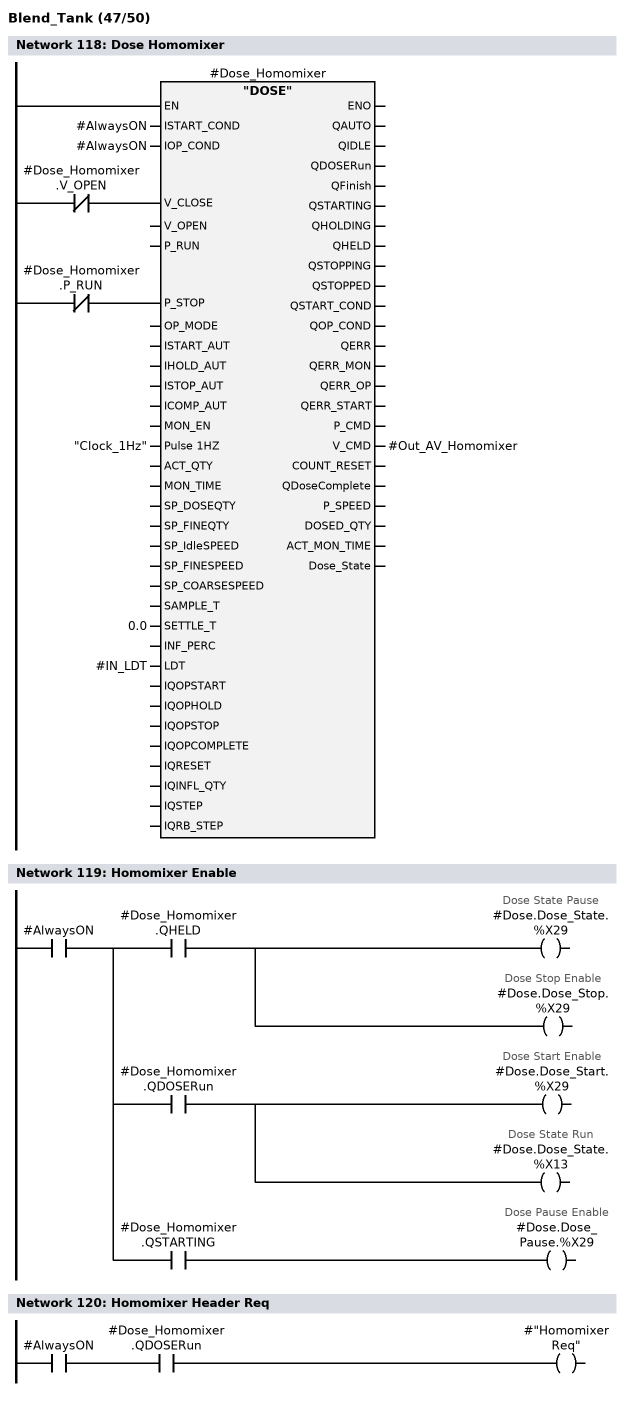
   RUNG wire#powerrail
      #Dose_Homomixer(V_CLOSE := wire#w1, P_STOP := wire#w2, ISTART_COND := #AlwaysON, IOP_COND := #AlwaysON, V_OPEN :=, P_RUN :=, OP_MODE :=, ISTART_AUT :=, IHOLD_AUT :=, ISTOP_AUT :=, ICOMP_AUT :=, MON_EN :=, "Pulse 1HZ" := "Clock_1Hz", ACT_QTY :=, MON_TIME :=, SP_DOSEQTY :=, SP_FINEQTY :=, SP_IdleSPEED :=, SP_FINESPEED :=, SP_COARSESPEED :=, SAMPLE_T :=, SETTLE_T := 0.0, INF_PERC :=, LDT := #IN_LDT, IQOPSTART :=, IQOPHOLD :=, IQOPSTOP :=, IQOPCOMPLETE :=, IQRESET :=, IQINFL_QTY :=, IQSTEP :=, IQRB_STEP :=, QAUTO =>, QIDLE =>, QDOSERun =>, QFinish =>, QSTARTING =>, QHOLDING =>, QHELD =>, QSTOPPING =>, QSTOPPED =>, QSTART_COND =>, QOP_COND =>, QERR =>, QERR_MON =>, QERR_OP =>, QERR_START =>, P_CMD =>, V_CMD => #Out_AV_Homomixer, COUNT_RESET =>, QDoseComplete =>, P_SPEED =>, DOSED_QTY =>, ACT_MON_TIME =>, Dose_State =>)
   END_RUNG
   RUNG wire#powerrail
      I_Contact( #Dose_Homomixer.V_OPEN )
   END_RUNG wire#w1
   RUNG wire#powerrail
      I_Contact( #Dose_Homomixer.P_RUN )
   END_RUNG wire#w2
   // the same network as SCL:
   #Dose_Homomixer(ISTART_COND := #AlwaysON,   // "DOSE"
                   IOP_COND := #AlwaysON,
                   V_CLOSE := NOT #Dose_Homomixer.V_OPEN,
                   P_STOP := NOT #Dose_Homomixer.P_RUN,
                   "Pulse 1HZ" := "Clock_1Hz",
                   SETTLE_T := 0.0,
                   LDT := #IN_LDT,
                   V_CMD => #Out_AV_Homomixer);
END_REGION

REGION Network 119: Homomixer Enable
   RUNG wire#powerrail
      Contact( #AlwaysON )
      wire#w1
      Contact( #Dose_Homomixer.QHELD )
      wire#w2
      Coil( #Dose.Dose_State.%X29 )   // Dose State Pause
   END_RUNG
   RUNG wire#w2
      Coil( #Dose.Dose_Stop.%X29 )   // Dose Stop Enable
   END_RUNG
   RUNG wire#w1
      Contact( #Dose_Homomixer.QDOSERun )
      wire#w3
      Coil( #Dose.Dose_Start.%X29 )   // Dose Start Enable
   END_RUNG
   RUNG wire#w3
      Coil( #Dose.Dose_State.%X13 )   // Dose State Run
   END_RUNG
   RUNG wire#w1
      Contact( #Dose_Homomixer.QSTARTING )
      Coil( #Dose.Dose_Pause.%X29 )   // Dose Pause Enable
   END_RUNG
   // the same network as SCL:
   #Dose.Dose_State.%X29 := #AlwaysON AND #Dose_Homomixer.QHELD;   // Dose State Pause
   #Dose.Dose_Stop.%X29 := #Dose.Dose_State.%X29;   // Dose Stop Enable
   #Dose.Dose_Start.%X29 := #AlwaysON AND #Dose_Homomixer.QDOSERun;   // Dose Start Enable
   #Dose.Dose_State.%X13 := #Dose.Dose_Start.%X29;   // Dose State Run
   #Dose.Dose_Pause.%X29 := #AlwaysON AND #Dose_Homomixer.QSTARTING;   // Dose Pause Enable
END_REGION

REGION Network 120: Homomixer Header Req
   RUNG wire#powerrail
      Contact( #AlwaysON )
      Contact( #Dose_Homomixer.QDOSERun )
      Coil( #"Homomixer Req" )
   END_RUNG
   // the same network as SCL:
   #"Homomixer Req" := #AlwaysON AND #Dose_Homomixer.QDOSERun;
END_REGION

REGION Network 122: Level Scaling
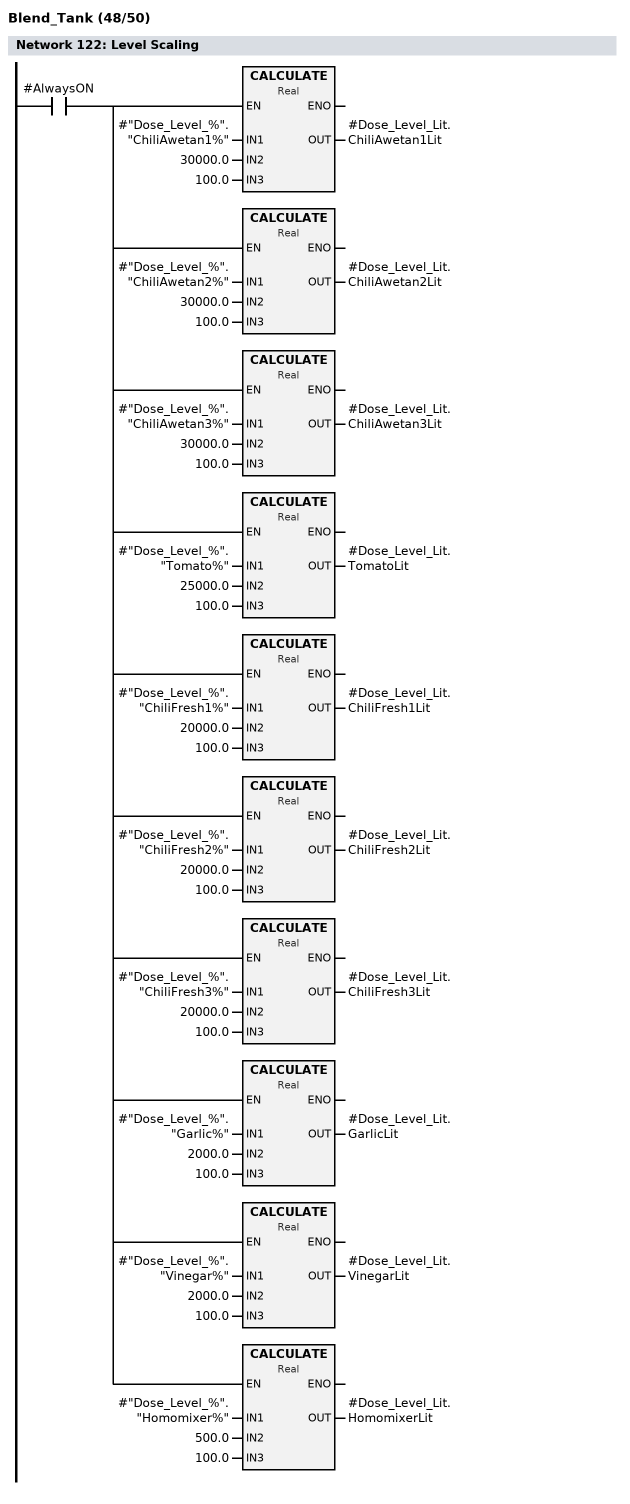
   RUNG wire#powerrail
      Contact( #AlwaysON )
      wire#w1
      { S7_Templates := "SrcType := Real"; S7_Expression := "(IN1 * IN2) / IN3" } Calculate(in1 := #"Dose_Level_%"."ChiliAwetan1%", in2 := 30000.0, in3 := 100.0, out => #Dose_Level_Lit.ChiliAwetan1Lit)
   END_RUNG
   RUNG wire#w1
      { S7_Templates := "SrcType := Real"; S7_Expression := "(IN1 * IN2) / IN3" } Calculate(in1 := #"Dose_Level_%"."ChiliAwetan2%", in2 := 30000.0, in3 := 100.0, out => #Dose_Level_Lit.ChiliAwetan2Lit)
   END_RUNG
   RUNG wire#w1
      { S7_Templates := "SrcType := Real"; S7_Expression := "(IN1 * IN2) / IN3" } Calculate(in1 := #"Dose_Level_%"."ChiliAwetan3%", in2 := 30000.0, in3 := 100.0, out => #Dose_Level_Lit.ChiliAwetan3Lit)
   END_RUNG
   RUNG wire#w1
      { S7_Templates := "SrcType := Real"; S7_Expression := "(IN1 * IN2) / IN3" } Calculate(in1 := #"Dose_Level_%"."Tomato%", in2 := 25000.0, in3 := 100.0, out => #Dose_Level_Lit.TomatoLit)
   END_RUNG
   RUNG wire#w1
      { S7_Templates := "SrcType := Real"; S7_Expression := "(IN1 * IN2) / IN3" } Calculate(in1 := #"Dose_Level_%"."ChiliFresh1%", in2 := 20000.0, in3 := 100.0, out => #Dose_Level_Lit.ChiliFresh1Lit)
   END_RUNG
   RUNG wire#w1
      { S7_Templates := "SrcType := Real"; S7_Expression := "(IN1 * IN2) / IN3" } Calculate(in1 := #"Dose_Level_%"."ChiliFresh2%", in2 := 20000.0, in3 := 100.0, out => #Dose_Level_Lit.ChiliFresh2Lit)
   END_RUNG
   RUNG wire#w1
      { S7_Templates := "SrcType := Real"; S7_Expression := "(IN1 * IN2) / IN3" } Calculate(in1 := #"Dose_Level_%"."ChiliFresh3%", in2 := 20000.0, in3 := 100.0, out => #Dose_Level_Lit.ChiliFresh3Lit)
   END_RUNG
   RUNG wire#w1
      { S7_Templates := "SrcType := Real"; S7_Expression := "(IN1 * IN2) / IN3" } Calculate(in1 := #"Dose_Level_%"."Garlic%", in2 := 2000.0, in3 := 100.0, out => #Dose_Level_Lit.GarlicLit)
   END_RUNG
   RUNG wire#w1
      { S7_Templates := "SrcType := Real"; S7_Expression := "(IN1 * IN2) / IN3" } Calculate(in1 := #"Dose_Level_%"."Vinegar%", in2 := 2000.0, in3 := 100.0, out => #Dose_Level_Lit.VinegarLit)
   END_RUNG
   RUNG wire#w1
      { S7_Templates := "SrcType := Real"; S7_Expression := "(IN1 * IN2) / IN3" } Calculate(in1 := #"Dose_Level_%"."Homomixer%", in2 := 500.0, in3 := 100.0, out => #Dose_Level_Lit.HomomixerLit)
   END_RUNG
   // the same network as SCL:
   IF #AlwaysON THEN
       #Dose_Level_Lit.ChiliAwetan1Lit := (#"Dose_Level_%"."ChiliAwetan1%" * 30000.0) / 100.0;
       #Dose_Level_Lit.ChiliAwetan2Lit := (#"Dose_Level_%"."ChiliAwetan2%" * 30000.0) / 100.0;
       #Dose_Level_Lit.ChiliAwetan3Lit := (#"Dose_Level_%"."ChiliAwetan3%" * 30000.0) / 100.0;
       #Dose_Level_Lit.TomatoLit := (#"Dose_Level_%"."Tomato%" * 25000.0) / 100.0;
       #Dose_Level_Lit.ChiliFresh1Lit := (#"Dose_Level_%"."ChiliFresh1%" * 20000.0) / 100.0;
       #Dose_Level_Lit.ChiliFresh2Lit := (#"Dose_Level_%"."ChiliFresh2%" * 20000.0) / 100.0;
       #Dose_Level_Lit.ChiliFresh3Lit := (#"Dose_Level_%"."ChiliFresh3%" * 20000.0) / 100.0;
       #Dose_Level_Lit.GarlicLit := (#"Dose_Level_%"."Garlic%" * 2000.0) / 100.0;
       #Dose_Level_Lit.VinegarLit := (#"Dose_Level_%"."Vinegar%" * 2000.0) / 100.0;
       #Dose_Level_Lit.HomomixerLit := (#"Dose_Level_%"."Homomixer%" * 500.0) / 100.0;
   END_IF;
END_REGION

REGION Network 123: Last Dose Qty
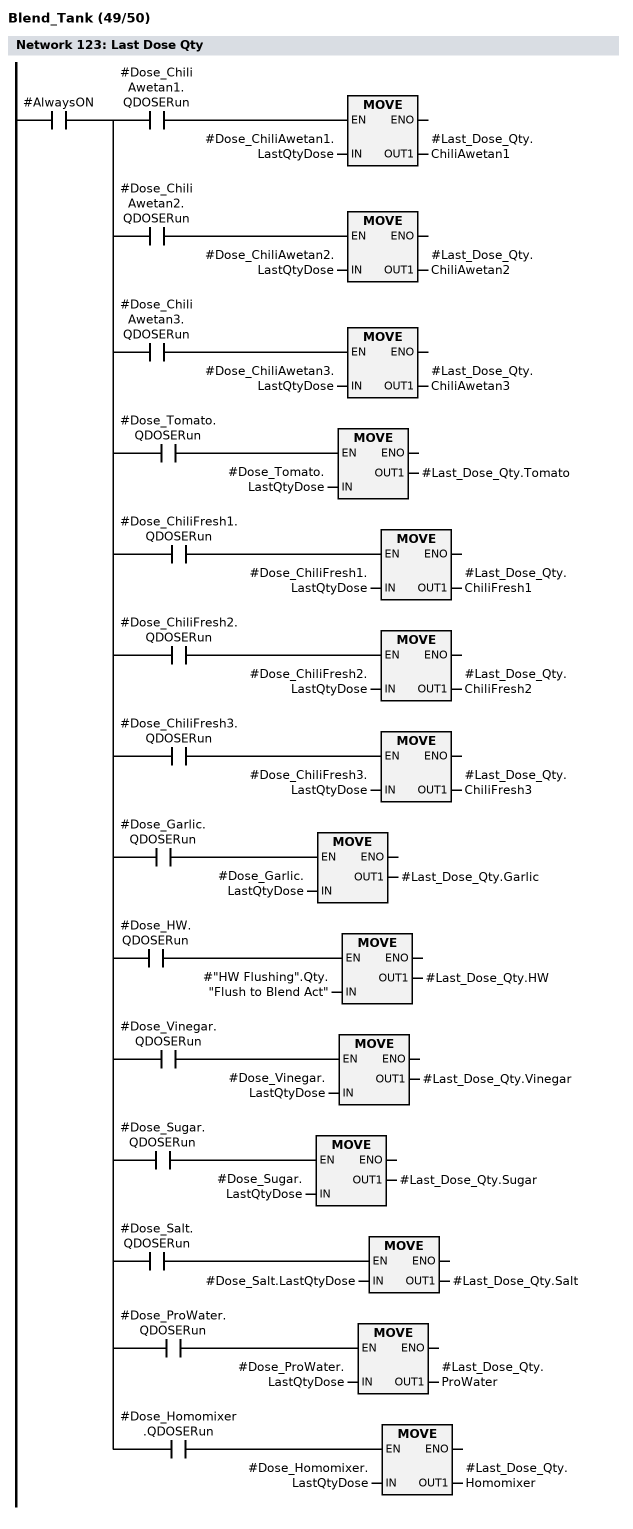
   RUNG wire#powerrail
      Contact( #AlwaysON )
      wire#w1
      Contact( #Dose_ChiliAwetan1.QDOSERun )
      Move(in := #Dose_ChiliAwetan1.LastQtyDose, out1 => #Last_Dose_Qty.ChiliAwetan1)
   END_RUNG
   RUNG wire#w1
      Contact( #Dose_ChiliAwetan2.QDOSERun )
      Move(in := #Dose_ChiliAwetan2.LastQtyDose, out1 => #Last_Dose_Qty.ChiliAwetan2)
   END_RUNG
   RUNG wire#w1
      Contact( #Dose_ChiliAwetan3.QDOSERun )
      Move(in := #Dose_ChiliAwetan3.LastQtyDose, out1 => #Last_Dose_Qty.ChiliAwetan3)
   END_RUNG
   RUNG wire#w1
      Contact( #Dose_Tomato.QDOSERun )
      Move(in := #Dose_Tomato.LastQtyDose, out1 => #Last_Dose_Qty.Tomato)
   END_RUNG
   RUNG wire#w1
      Contact( #Dose_ChiliFresh1.QDOSERun )
      Move(in := #Dose_ChiliFresh1.LastQtyDose, out1 => #Last_Dose_Qty.ChiliFresh1)
   END_RUNG
   RUNG wire#w1
      Contact( #Dose_ChiliFresh2.QDOSERun )
      Move(in := #Dose_ChiliFresh2.LastQtyDose, out1 => #Last_Dose_Qty.ChiliFresh2)
   END_RUNG
   RUNG wire#w1
      Contact( #Dose_ChiliFresh3.QDOSERun )
      Move(in := #Dose_ChiliFresh3.LastQtyDose, out1 => #Last_Dose_Qty.ChiliFresh3)
   END_RUNG
   RUNG wire#w1
      Contact( #Dose_Garlic.QDOSERun )
      Move(in := #Dose_Garlic.LastQtyDose, out1 => #Last_Dose_Qty.Garlic)
   END_RUNG
   RUNG wire#w1
      Contact( #Dose_HW.QDOSERun )
      Move(in := #"HW Flushing".Qty."Flush to Blend Act", out1 => #Last_Dose_Qty.HW)
   END_RUNG
   RUNG wire#w1
      Contact( #Dose_Vinegar.QDOSERun )
      Move(in := #Dose_Vinegar.LastQtyDose, out1 => #Last_Dose_Qty.Vinegar)
   END_RUNG
   RUNG wire#w1
      Contact( #Dose_Sugar.QDOSERun )
      Move(in := #Dose_Sugar.LastQtyDose, out1 => #Last_Dose_Qty.Sugar)
   END_RUNG
   RUNG wire#w1
      Contact( #Dose_Salt.QDOSERun )
      Move(in := #Dose_Salt.LastQtyDose, out1 => #Last_Dose_Qty.Salt)
   END_RUNG
   RUNG wire#w1
      Contact( #Dose_ProWater.QDOSERun )
      Move(in := #Dose_ProWater.LastQtyDose, out1 => #Last_Dose_Qty.ProWater)
   END_RUNG
   RUNG wire#w1
      Contact( #Dose_Homomixer.QDOSERun )
      Move(in := #Dose_Homomixer.LastQtyDose, out1 => #Last_Dose_Qty.Homomixer)
   END_RUNG
   // the same network as SCL:
   IF #AlwaysON AND #Dose_ChiliAwetan1.QDOSERun THEN
       #Last_Dose_Qty.ChiliAwetan1 := #Dose_ChiliAwetan1.LastQtyDose;
   END_IF;
   IF #AlwaysON AND #Dose_ChiliAwetan2.QDOSERun THEN
       #Last_Dose_Qty.ChiliAwetan2 := #Dose_ChiliAwetan2.LastQtyDose;
   END_IF;
   IF #AlwaysON AND #Dose_ChiliAwetan3.QDOSERun THEN
       #Last_Dose_Qty.ChiliAwetan3 := #Dose_ChiliAwetan3.LastQtyDose;
   END_IF;
   IF #AlwaysON AND #Dose_Tomato.QDOSERun THEN #Last_Dose_Qty.Tomato := #Dose_Tomato.LastQtyDose; END_IF;
   IF #AlwaysON AND #Dose_ChiliFresh1.QDOSERun THEN
       #Last_Dose_Qty.ChiliFresh1 := #Dose_ChiliFresh1.LastQtyDose;
   END_IF;
   IF #AlwaysON AND #Dose_ChiliFresh2.QDOSERun THEN
       #Last_Dose_Qty.ChiliFresh2 := #Dose_ChiliFresh2.LastQtyDose;
   END_IF;
   IF #AlwaysON AND #Dose_ChiliFresh3.QDOSERun THEN
       #Last_Dose_Qty.ChiliFresh3 := #Dose_ChiliFresh3.LastQtyDose;
   END_IF;
   IF #AlwaysON AND #Dose_Garlic.QDOSERun THEN #Last_Dose_Qty.Garlic := #Dose_Garlic.LastQtyDose; END_IF;
   IF #AlwaysON AND #Dose_HW.QDOSERun THEN
       #Last_Dose_Qty.HW := #"HW Flushing".Qty."Flush to Blend Act";
   END_IF;
   IF #AlwaysON AND #Dose_Vinegar.QDOSERun THEN #Last_Dose_Qty.Vinegar := #Dose_Vinegar.LastQtyDose; END_IF;
   IF #AlwaysON AND #Dose_Sugar.QDOSERun THEN #Last_Dose_Qty.Sugar := #Dose_Sugar.LastQtyDose; END_IF;
   IF #AlwaysON AND #Dose_Salt.QDOSERun THEN #Last_Dose_Qty.Salt := #Dose_Salt.LastQtyDose; END_IF;
   IF #AlwaysON AND #Dose_ProWater.QDOSERun THEN
       #Last_Dose_Qty.ProWater := #Dose_ProWater.LastQtyDose;
   END_IF;
   IF #AlwaysON AND #Dose_Homomixer.QDOSERun THEN
       #Last_Dose_Qty.Homomixer := #Dose_Homomixer.LastQtyDose;
   END_IF;
END_REGION

REGION Network 124: Reset Last Dose Qty After CIP Tank
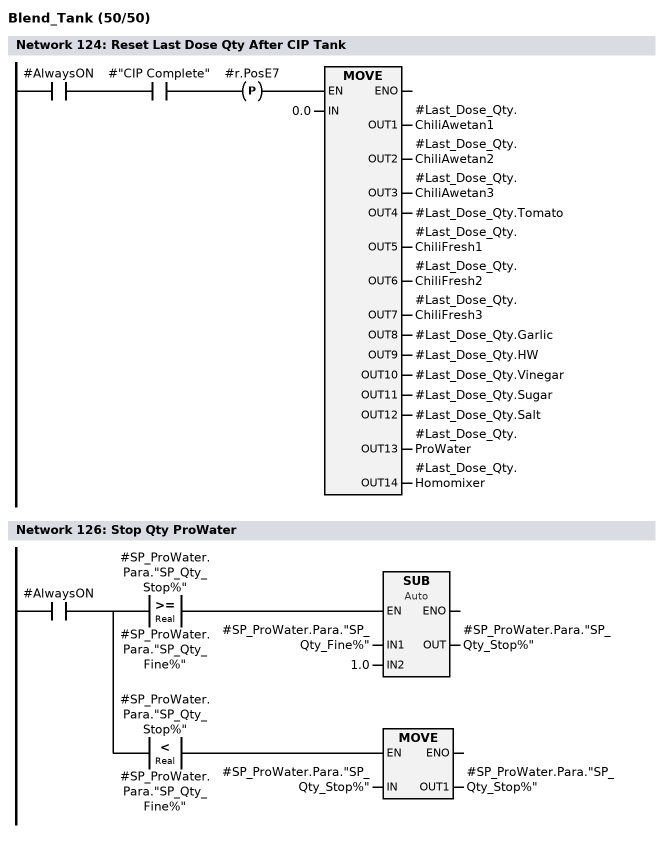
   RUNG wire#powerrail
      Contact( #AlwaysON )
      Contact( #"CIP Complete" )
      P_Trig( #r.PosE7 )
      Move(in := 0.0, out1 => #Last_Dose_Qty.ChiliAwetan1, out2 => #Last_Dose_Qty.ChiliAwetan2, out3 => #Last_Dose_Qty.ChiliAwetan3, out4 => #Last_Dose_Qty.Tomato, out5 => #Last_Dose_Qty.ChiliFresh1, out6 => #Last_Dose_Qty.ChiliFresh2, out7 => #Last_Dose_Qty.ChiliFresh3, out8 => #Last_Dose_Qty.Garlic, out9 => #Last_Dose_Qty.HW, out10 => #Last_Dose_Qty.Vinegar, out11 => #Last_Dose_Qty.Sugar, out12 => #Last_Dose_Qty.Salt, out13 => #Last_Dose_Qty.ProWater, out14 => #Last_Dose_Qty.Homomixer)
   END_RUNG
   // the same network as SCL:
   #_w1 := #AlwaysON AND #"CIP Complete";
   #_w2 := #_w1 AND NOT #r.PosE7;   // rising edge
   #r.PosE7 := #_w1;
   IF #_w2 THEN
       #Last_Dose_Qty.ChiliAwetan1 := 0.0;
       #Last_Dose_Qty.ChiliAwetan2 := 0.0;
       #Last_Dose_Qty.ChiliAwetan3 := 0.0;
       #Last_Dose_Qty.Tomato := 0.0;
       #Last_Dose_Qty.ChiliFresh1 := 0.0;
       #Last_Dose_Qty.ChiliFresh2 := 0.0;
       #Last_Dose_Qty.ChiliFresh3 := 0.0;
       #Last_Dose_Qty.Garlic := 0.0;
       #Last_Dose_Qty.HW := 0.0;
       #Last_Dose_Qty.Vinegar := 0.0;
       #Last_Dose_Qty.Sugar := 0.0;
       #Last_Dose_Qty.Salt := 0.0;
       #Last_Dose_Qty.ProWater := 0.0;
       #Last_Dose_Qty.Homomixer := 0.0;
   END_IF;
END_REGION

REGION Network 126: Stop Qty ProWater
   RUNG wire#powerrail
      Contact( #AlwaysON )
      wire#w1
      { S7_Templates := "SrcType := Real" } GE_Contact(in1 := #SP_ProWater.Para."SP_Qty_Stop%", in2 := #SP_ProWater.Para."SP_Qty_Fine%")
      Sub(in1 := #SP_ProWater.Para."SP_Qty_Fine%", in2 := 1.0, out => #SP_ProWater.Para."SP_Qty_Stop%")
   END_RUNG
   RUNG wire#w1
      { S7_Templates := "SrcType := Real" } LT_Contact(in1 := #SP_ProWater.Para."SP_Qty_Stop%", in2 := #SP_ProWater.Para."SP_Qty_Fine%")
      Move(in := #SP_ProWater.Para."SP_Qty_Stop%", out1 => #SP_ProWater.Para."SP_Qty_Stop%")
   END_RUNG
   // the same network as SCL:
   IF #AlwaysON AND (#SP_ProWater.Para."SP_Qty_Stop%" >= #SP_ProWater.Para."SP_Qty_Fine%") THEN
       #SP_ProWater.Para."SP_Qty_Stop%" := #SP_ProWater.Para."SP_Qty_Fine%" - 1.0;
   END_IF;
   IF #AlwaysON AND (#SP_ProWater.Para."SP_Qty_Stop%" < #SP_ProWater.Para."SP_Qty_Fine%") THEN
       #SP_ProWater.Para."SP_Qty_Stop%" := #SP_ProWater.Para."SP_Qty_Stop%";
   END_IF;
END_REGION
END_FUNCTION_BLOCK

FUNCTION_BLOCK "IO_Valve_Blend20"   // FB24, LAD
{ S7_Optimized_Access := 'FALSE' }
VERSION : 0.1
// stored: AutoNumber true, IsIECCheckEnabled false, SetENOAutomatically false, UDAEnableTagReadback false
   VAR_INPUT
      "lock 1" : Bool;
      "lock 2" : Bool;
      "lock 3" : Bool;
      "lock 4" : Bool;
      init : Bool;
      reset : Bool;
      testing : Bool;
   END_VAR
   VAR
      "AV-20.01" : "Valve";
      "AV-20.02" : "Valve";
      "AV-20.03" : "Valve";
      "AV-20.04" : "Valve";
      "AV-20.05" : "Valve";
      "AV-20.06" : "Valve";
      "AV-20.07" : "Valve";
      "AV-20.08" : "Valve";
      "AV-20.09" : "Valve";
      "AV-20.10" : "Valve";
      "AV-20.11" : "Valve";
      "AV-20.21" : "Valve";
      "AV-20.22" : "Valve";
      "AV-20.23" : "Valve";
      "AV-20.24" : "Valve";
      "AV-20.25" : "Valve";
      "AV-20.26" : "Valve";
      "AV-20.27" : "Valve";
      "AV-20.28" : "Valve";
      "AV-20.29" : "Valve";
      "AV-20.30" : "Valve";
      "AV-20.31" : "Valve";
      "AV-20.32" : "Valve";
      "AV-20.33" : "Valve";
      "AV-20.34" : "Valve";
      "AV-20.35" : "Valve";
      "AV-20.36" : "Valve";
      "AV-20.37" : "Valve";
      "AV-20.41" : "Valve";
      "AV-20.42" : "Valve";
   END_VAR
BEGIN

REGION Network 1 (SCL): FB OPEN AND CLOSE VALVE T-20
   IF #testing THEN
       // Statement section IF
       #"AV-20.01".FB_OPEN := #"AV-20.01".QCMD_OP;
       #"AV-20.01".FB_CLOSE := NOT #"AV-20.01".QCMD_OP;
       #"AV-20.02".FB_OPEN := #"AV-20.02".QCMD_OP;
       #"AV-20.02".FB_CLOSE := NOT #"AV-20.02".QCMD_OP;
       #"AV-20.03".FB_OPEN := #"AV-20.03".QCMD_OP;
       #"AV-20.03".FB_CLOSE := NOT #"AV-20.03".QCMD_OP;
       #"AV-20.04".FB_OPEN := #"AV-20.04".QCMD_OP;
       #"AV-20.04".FB_CLOSE := NOT #"AV-20.04".QCMD_OP;
       #"AV-20.05".FB_OPEN := #"AV-20.05".QCMD_OP;
       #"AV-20.05".FB_CLOSE := NOT #"AV-20.05".QCMD_OP;
       #"AV-20.06".FB_OPEN := #"AV-20.06".QCMD_OP;
       #"AV-20.06".FB_CLOSE := NOT #"AV-20.06".QCMD_OP;
       #"AV-20.07".FB_OPEN := #"AV-20.07".QCMD_OP;
       #"AV-20.07".FB_CLOSE := NOT #"AV-20.07".QCMD_OP;
       #"AV-20.08".FB_OPEN := #"AV-20.08".QCMD_OP;
       #"AV-20.08".FB_CLOSE := NOT #"AV-20.08".QCMD_OP;
       #"AV-20.09".FB_OPEN := #"AV-20.09".QCMD_OP;
       #"AV-20.09".FB_CLOSE := NOT #"AV-20.09".QCMD_OP;
       #"AV-20.10".FB_OPEN := #"AV-20.10".QCMD_OP;
       #"AV-20.10".FB_CLOSE := NOT #"AV-20.10".QCMD_OP;
       #"AV-20.11".FB_OPEN := #"AV-20.11".QCMD_OP;
       #"AV-20.11".FB_CLOSE := NOT #"AV-20.11".QCMD_OP;
       #"AV-20.21".FB_OPEN := #"AV-20.21".QCMD_OP;
       #"AV-20.21".FB_CLOSE := NOT #"AV-20.21".QCMD_OP;
       #"AV-20.22".FB_OPEN := #"AV-20.22".QCMD_OP;
       #"AV-20.22".FB_CLOSE := NOT #"AV-20.22".QCMD_OP;
       #"AV-20.23".FB_OPEN := #"AV-20.23".QCMD_OP;
       #"AV-20.23".FB_CLOSE := NOT #"AV-20.23".QCMD_OP;
       #"AV-20.24".FB_OPEN := #"AV-20.24".QCMD_OP;
       #"AV-20.24".FB_CLOSE := NOT #"AV-20.24".QCMD_OP;
       #"AV-20.25".FB_OPEN := #"AV-20.25".QCMD_OP;
       #"AV-20.25".FB_CLOSE := NOT #"AV-20.25".QCMD_OP;
       #"AV-20.26".FB_OPEN := #"AV-20.26".QCMD_OP;
       #"AV-20.26".FB_CLOSE := NOT #"AV-20.26".QCMD_OP;
       #"AV-20.27".FB_OPEN := #"AV-20.27".QCMD_OP;
       #"AV-20.27".FB_CLOSE := NOT #"AV-20.27".QCMD_OP;
       #"AV-20.28".FB_OPEN := #"AV-20.28".QCMD_OP;
       #"AV-20.28".FB_CLOSE := NOT #"AV-20.28".QCMD_OP;
       #"AV-20.29".FB_OPEN := #"AV-20.29".QCMD_OP;
       #"AV-20.29".FB_CLOSE := NOT #"AV-20.29".QCMD_OP;
       #"AV-20.30".FB_OPEN := #"AV-20.30".QCMD_OP;
       #"AV-20.30".FB_CLOSE := NOT #"AV-20.30".QCMD_OP;
       #"AV-20.31".FB_OPEN := #"AV-20.31".QCMD_OP;
       #"AV-20.31".FB_CLOSE := NOT #"AV-20.31".QCMD_OP;
       #"AV-20.32".FB_OPEN := #"AV-20.32".QCMD_OP;
       #"AV-20.32".FB_CLOSE := NOT #"AV-20.32".QCMD_OP;
       #"AV-20.33".FB_OPEN := #"AV-20.33".QCMD_OP;
       #"AV-20.33".FB_CLOSE := NOT #"AV-20.33".QCMD_OP;
       #"AV-20.34".FB_OPEN := #"AV-20.34".QCMD_OP;
       #"AV-20.34".FB_CLOSE := NOT #"AV-20.34".QCMD_OP;
       #"AV-20.35".FB_OPEN := #"AV-20.35".QCMD_OP;
       #"AV-20.35".FB_CLOSE := NOT #"AV-20.35".QCMD_OP;
       #"AV-20.36".FB_OPEN := #"AV-20.36".QCMD_OP;
       #"AV-20.36".FB_CLOSE := NOT #"AV-20.36".QCMD_OP;
       #"AV-20.37".FB_OPEN := #"AV-20.37".QCMD_OP;
       #"AV-20.37".FB_CLOSE := NOT #"AV-20.37".QCMD_OP;
       #"AV-20.41".FB_OPEN := #"AV-20.41".QCMD_OP;
       #"AV-20.41".FB_CLOSE := NOT #"AV-20.41".QCMD_OP;
       #"AV-20.42".FB_OPEN := #"AV-20.42".QCMD_OP;
       #"AV-20.42".FB_CLOSE := NOT #"AV-20.42".QCMD_OP;
   ELSE
       // Statement section ELSE
       #"AV-20.01".FB_OPEN := #"AV-20.01".QCMD_OP;
       #"AV-20.01".FB_CLOSE := NOT #"AV-20.01".QCMD_OP;
       #"AV-20.02".FB_OPEN := NOT "ZSC-20.02";
       #"AV-20.02".FB_CLOSE := "ZSC-20.02";
       #"AV-20.03".FB_OPEN := NOT "ZSC-20.03";
       #"AV-20.03".FB_CLOSE := "ZSC-20.03";
       #"AV-20.04".FB_OPEN := #"AV-20.04".QCMD_OP;
       #"AV-20.04".FB_CLOSE := NOT #"AV-20.04".QCMD_OP;
       #"AV-20.05".FB_OPEN := NOT "ZSC-20.05";
       #"AV-20.05".FB_CLOSE := "ZSC-20.05";
       #"AV-20.06".FB_OPEN := NOT "ZSC-20.06";
       #"AV-20.06".FB_CLOSE := "ZSC-20.06";
       #"AV-20.07".FB_OPEN := #"AV-20.07".QCMD_OP;
       #"AV-20.07".FB_CLOSE := NOT #"AV-20.07".QCMD_OP;
       #"AV-20.08".FB_OPEN := NOT "ZSC-20.08";
       #"AV-20.08".FB_CLOSE := "ZSC-20.08";
       #"AV-20.09".FB_OPEN := NOT "ZSC-20.09";
       #"AV-20.09".FB_CLOSE := "ZSC-20.09";
       #"AV-20.10".FB_OPEN := #"AV-20.10".QCMD_OP;
       #"AV-20.10".FB_CLOSE := NOT #"AV-20.10".QCMD_OP;
       #"AV-20.11".FB_OPEN := NOT "ZSC-20.11";
       #"AV-20.11".FB_CLOSE := "ZSC-20.11";
       #"AV-20.21".FB_OPEN := NOT "ZSC-20.21";
       #"AV-20.21".FB_CLOSE := "ZSC-20.21";
       #"AV-20.22".FB_OPEN := #"AV-20.22".QCMD_OP;
       #"AV-20.22".FB_CLOSE := NOT #"AV-20.22".QCMD_OP;
       #"AV-20.23".FB_OPEN := NOT "ZSC-20.23";
       #"AV-20.23".FB_CLOSE := "ZSC-20.23";
       #"AV-20.24".FB_OPEN := NOT "ZSC-20.24";
       #"AV-20.24".FB_CLOSE := "ZSC-20.24";
       #"AV-20.25".FB_OPEN := NOT "ZSC-20.25";
       #"AV-20.25".FB_CLOSE := "ZSC-20.25";
       #"AV-20.26".FB_OPEN := #"AV-20.26".QCMD_OP;
       #"AV-20.26".FB_CLOSE := NOT #"AV-20.26".QCMD_OP;
       #"AV-20.27".FB_OPEN := NOT "ZSC-20.27";
       #"AV-20.27".FB_CLOSE := "ZSC-20.27";
       #"AV-20.28".FB_OPEN := NOT "ZSC-20.28";
       #"AV-20.28".FB_CLOSE := "ZSC-20.28";
       #"AV-20.29".FB_OPEN := #"AV-20.29".QCMD_OP;
       #"AV-20.29".FB_CLOSE := NOT #"AV-20.29".QCMD_OP;
       #"AV-20.30".FB_OPEN := #"AV-20.30".QCMD_OP;
       #"AV-20.30".FB_CLOSE := NOT #"AV-20.30".QCMD_OP;
       #"AV-20.31".FB_OPEN := NOT "ZSC-20.31";
       #"AV-20.31".FB_CLOSE := "ZSC-20.31";
       #"AV-20.32".FB_OPEN := NOT "ZSC-20.32";
       #"AV-20.32".FB_CLOSE := "ZSC-20.32";
       #"AV-20.33".FB_OPEN := NOT "ZSC-20.33";
       #"AV-20.33".FB_CLOSE := "ZSC-20.33";
       #"AV-20.34".FB_OPEN := NOT "ZSC-20.34";
       #"AV-20.34".FB_CLOSE := "ZSC-20.34";
       #"AV-20.35".FB_OPEN := NOT "ZSC-20.35";
       #"AV-20.35".FB_CLOSE := "ZSC-20.35";
       #"AV-20.36".FB_OPEN := NOT "ZSC-20.36";
       #"AV-20.36".FB_CLOSE := "ZSC-20.36";
       #"AV-20.37".FB_OPEN := NOT "ZSC-20.37";
       #"AV-20.37".FB_CLOSE := "ZSC-20.37";
       #"AV-20.41".FB_OPEN := #"AV-20.41".QCMD_OP;
       #"AV-20.41".FB_CLOSE := NOT #"AV-20.41".QCMD_OP;
       #"AV-20.42".FB_OPEN := #"AV-20.42".QCMD_OP;
       #"AV-20.42".FB_CLOSE := NOT #"AV-20.42".QCMD_OP;
   END_IF;
END_REGION

NETWORK
TITLE = FB MONITORING TIME VALVE T-20
// FB OPEN TIME
      L     T#20s;
      T     #"AV-20.01".MON_T;
      T     #"AV-20.02".MON_T;
      T     #"AV-20.03".MON_T;
      T     #"AV-20.04".MON_T;
      T     #"AV-20.05".MON_T;
      T     #"AV-20.06".MON_T;
      T     #"AV-20.07".MON_T;
      T     #"AV-20.08".MON_T;
      T     #"AV-20.09".MON_T;
      T     #"AV-20.10".MON_T;
      T     #"AV-20.11".MON_T;
      T     #"AV-20.21".MON_T;
      T     #"AV-20.22".MON_T;
      T     #"AV-20.23".MON_T;
      T     #"AV-20.24".MON_T;
      T     #"AV-20.25".MON_T;
      T     #"AV-20.26".MON_T;
      T     #"AV-20.27".MON_T;
      T     #"AV-20.28".MON_T;
      T     #"AV-20.29".MON_T;
      T     #"AV-20.30".MON_T;
      T     #"AV-20.31".MON_T;
      T     #"AV-20.32".MON_T;
      T     #"AV-20.33".MON_T;
      T     #"AV-20.34".MON_T;
      T     #"AV-20.35".MON_T;
      T     #"AV-20.36".MON_T;
      T     #"AV-20.37".MON_T;
      T     #"AV-20.41".MON_T;
      T     #"AV-20.42".MON_T;

// FB CLOSE TIME
      L     T#20s;
      T     #"AV-20.01".MON_T_CLOSE;
      T     #"AV-20.02".MON_T_CLOSE;
      T     #"AV-20.03".MON_T_CLOSE;
      T     #"AV-20.04".MON_T_CLOSE;
      T     #"AV-20.05".MON_T_CLOSE;
      T     #"AV-20.06".MON_T_CLOSE;
      T     #"AV-20.07".MON_T_CLOSE;
      T     #"AV-20.08".MON_T_CLOSE;
      T     #"AV-20.09".MON_T_CLOSE;
      T     #"AV-20.10".MON_T_CLOSE;
      T     #"AV-20.11".MON_T_CLOSE;
      T     #"AV-20.21".MON_T_CLOSE;
      T     #"AV-20.22".MON_T_CLOSE;
      T     #"AV-20.23".MON_T_CLOSE;
      T     #"AV-20.24".MON_T_CLOSE;
      T     #"AV-20.25".MON_T_CLOSE;
      T     #"AV-20.26".MON_T_CLOSE;
      T     #"AV-20.27".MON_T_CLOSE;
      T     #"AV-20.28".MON_T_CLOSE;
      T     #"AV-20.29".MON_T_CLOSE;
      T     #"AV-20.30".MON_T_CLOSE;
      T     #"AV-20.31".MON_T_CLOSE;
      T     #"AV-20.32".MON_T_CLOSE;
      T     #"AV-20.33".MON_T_CLOSE;
      T     #"AV-20.34".MON_T_CLOSE;
      T     #"AV-20.35".MON_T_CLOSE;
      T     #"AV-20.36".MON_T_CLOSE;
      T     #"AV-20.37".MON_T_CLOSE;
      T     #"AV-20.41".MON_T_CLOSE;
      T     #"AV-20.42".MON_T_CLOSE;


REGION Network 3: AV-20.01
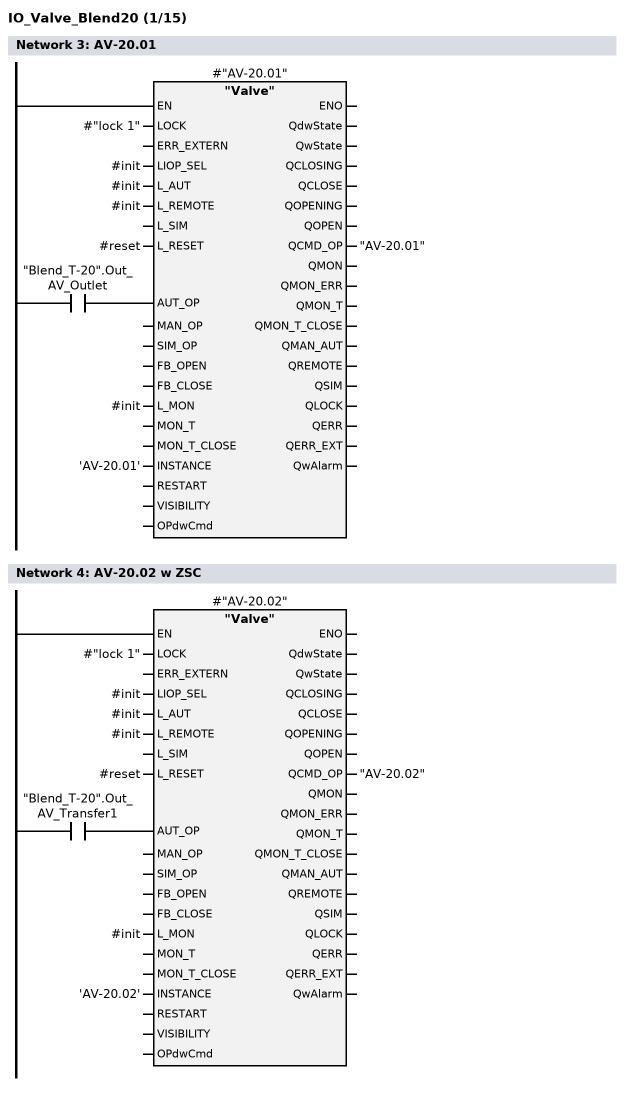
   RUNG wire#powerrail
      #"AV-20.01"(AUT_OP := wire#w1, LOCK := #"lock 1", ERR_EXTERN :=, LIOP_SEL := #init, L_AUT := #init, L_REMOTE := #init, L_SIM :=, L_RESET := #reset, MAN_OP :=, SIM_OP :=, FB_OPEN :=, FB_CLOSE :=, L_MON := #init, MON_T :=, MON_T_CLOSE :=, INSTANCE := 'AV-20.01', RESTART :=, VISIBILITY :=, OPdwCmd :=, QdwState =>, QwState =>, QCLOSING =>, QCLOSE =>, QOPENING =>, QOPEN =>, QCMD_OP => "AV-20.01", QMON =>, QMON_ERR =>, QMON_T =>, QMON_T_CLOSE =>, QMAN_AUT =>, QREMOTE =>, QSIM =>, QLOCK =>, QERR =>, QERR_EXT =>, QwAlarm =>)
   END_RUNG
   RUNG wire#powerrail
      Contact( "Blend_T-20".Out_AV_Outlet )
   END_RUNG wire#w1
   // the same network as SCL:
   #"AV-20.01"(LOCK := #"lock 1",   // "Valve"
               LIOP_SEL := #init,
               L_AUT := #init,
               L_REMOTE := #init,
               L_RESET := #reset,
               AUT_OP := "Blend_T-20".Out_AV_Outlet,
               L_MON := #init,
               INSTANCE := 'AV-20.01',
               QCMD_OP => "AV-20.01");
END_REGION

REGION Network 4: AV-20.02 w ZSC
   RUNG wire#powerrail
      #"AV-20.02"(AUT_OP := wire#w1, LOCK := #"lock 1", ERR_EXTERN :=, LIOP_SEL := #init, L_AUT := #init, L_REMOTE := #init, L_SIM :=, L_RESET := #reset, MAN_OP :=, SIM_OP :=, FB_OPEN :=, FB_CLOSE :=, L_MON := #init, MON_T :=, MON_T_CLOSE :=, INSTANCE := 'AV-20.02', RESTART :=, VISIBILITY :=, OPdwCmd :=, QdwState =>, QwState =>, QCLOSING =>, QCLOSE =>, QOPENING =>, QOPEN =>, QCMD_OP => "AV-20.02", QMON =>, QMON_ERR =>, QMON_T =>, QMON_T_CLOSE =>, QMAN_AUT =>, QREMOTE =>, QSIM =>, QLOCK =>, QERR =>, QERR_EXT =>, QwAlarm =>)
   END_RUNG
   RUNG wire#powerrail
      Contact( "Blend_T-20".Out_AV_Transfer1 )
   END_RUNG wire#w1
   // the same network as SCL:
   #"AV-20.02"(LOCK := #"lock 1",   // "Valve"
               LIOP_SEL := #init,
               L_AUT := #init,
               L_REMOTE := #init,
               L_RESET := #reset,
               AUT_OP := "Blend_T-20".Out_AV_Transfer1,
               L_MON := #init,
               INSTANCE := 'AV-20.02',
               QCMD_OP => "AV-20.02");
END_REGION

REGION Network 5: AV-20.03 w ZSC
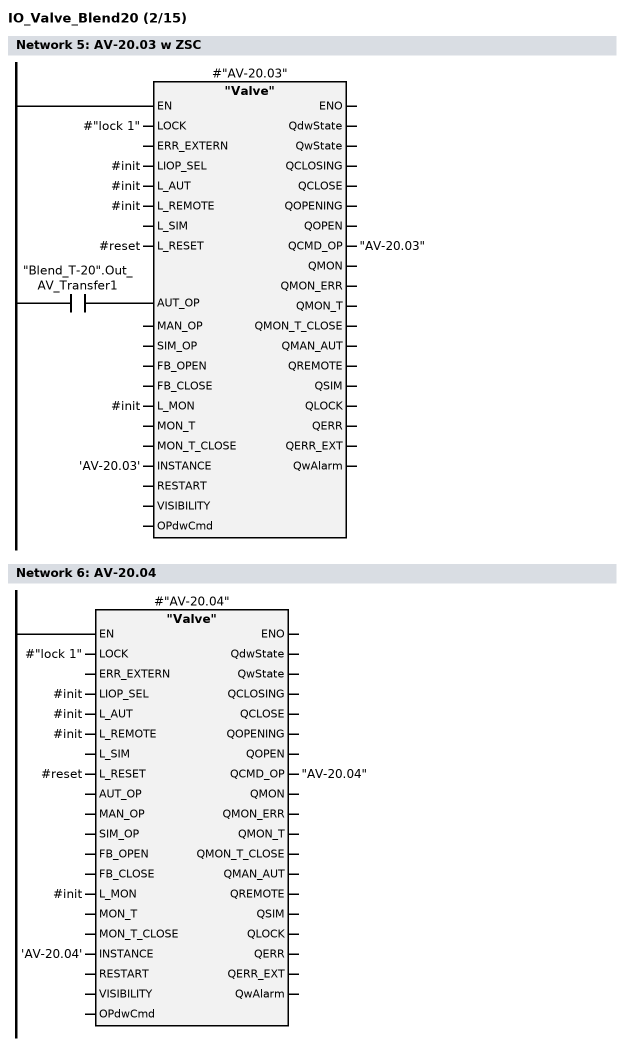
   RUNG wire#powerrail
      #"AV-20.03"(AUT_OP := wire#w1, LOCK := #"lock 1", ERR_EXTERN :=, LIOP_SEL := #init, L_AUT := #init, L_REMOTE := #init, L_SIM :=, L_RESET := #reset, MAN_OP :=, SIM_OP :=, FB_OPEN :=, FB_CLOSE :=, L_MON := #init, MON_T :=, MON_T_CLOSE :=, INSTANCE := 'AV-20.03', RESTART :=, VISIBILITY :=, OPdwCmd :=, QdwState =>, QwState =>, QCLOSING =>, QCLOSE =>, QOPENING =>, QOPEN =>, QCMD_OP => "AV-20.03", QMON =>, QMON_ERR =>, QMON_T =>, QMON_T_CLOSE =>, QMAN_AUT =>, QREMOTE =>, QSIM =>, QLOCK =>, QERR =>, QERR_EXT =>, QwAlarm =>)
   END_RUNG
   RUNG wire#powerrail
      Contact( "Blend_T-20".Out_AV_Transfer1 )
   END_RUNG wire#w1
   // the same network as SCL:
   #"AV-20.03"(LOCK := #"lock 1",   // "Valve"
               LIOP_SEL := #init,
               L_AUT := #init,
               L_REMOTE := #init,
               L_RESET := #reset,
               AUT_OP := "Blend_T-20".Out_AV_Transfer1,
               L_MON := #init,
               INSTANCE := 'AV-20.03',
               QCMD_OP => "AV-20.03");
END_REGION

REGION Network 6: AV-20.04
   RUNG wire#powerrail
      #"AV-20.04"(LOCK := #"lock 1", ERR_EXTERN :=, LIOP_SEL := #init, L_AUT := #init, L_REMOTE := #init, L_SIM :=, L_RESET := #reset, AUT_OP :=, MAN_OP :=, SIM_OP :=, FB_OPEN :=, FB_CLOSE :=, L_MON := #init, MON_T :=, MON_T_CLOSE :=, INSTANCE := 'AV-20.04', RESTART :=, VISIBILITY :=, OPdwCmd :=, QdwState =>, QwState =>, QCLOSING =>, QCLOSE =>, QOPENING =>, QOPEN =>, QCMD_OP => "AV-20.04", QMON =>, QMON_ERR =>, QMON_T =>, QMON_T_CLOSE =>, QMAN_AUT =>, QREMOTE =>, QSIM =>, QLOCK =>, QERR =>, QERR_EXT =>, QwAlarm =>)
   END_RUNG
   // the same network as SCL:
   #"AV-20.04"(LOCK := #"lock 1",   // "Valve"
               LIOP_SEL := #init,
               L_AUT := #init,
               L_REMOTE := #init,
               L_RESET := #reset,
               L_MON := #init,
               INSTANCE := 'AV-20.04',
               QCMD_OP => "AV-20.04");
END_REGION

REGION Network 7: AV-20.05 w ZSC
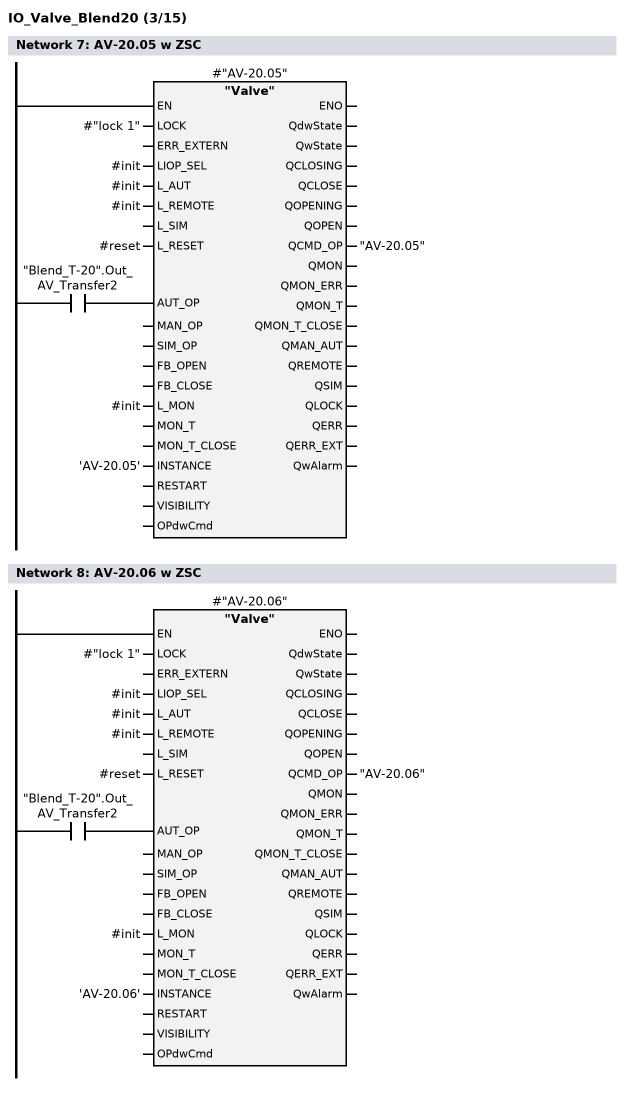
   RUNG wire#powerrail
      #"AV-20.05"(AUT_OP := wire#w1, LOCK := #"lock 1", ERR_EXTERN :=, LIOP_SEL := #init, L_AUT := #init, L_REMOTE := #init, L_SIM :=, L_RESET := #reset, MAN_OP :=, SIM_OP :=, FB_OPEN :=, FB_CLOSE :=, L_MON := #init, MON_T :=, MON_T_CLOSE :=, INSTANCE := 'AV-20.05', RESTART :=, VISIBILITY :=, OPdwCmd :=, QdwState =>, QwState =>, QCLOSING =>, QCLOSE =>, QOPENING =>, QOPEN =>, QCMD_OP => "AV-20.05", QMON =>, QMON_ERR =>, QMON_T =>, QMON_T_CLOSE =>, QMAN_AUT =>, QREMOTE =>, QSIM =>, QLOCK =>, QERR =>, QERR_EXT =>, QwAlarm =>)
   END_RUNG
   RUNG wire#powerrail
      Contact( "Blend_T-20".Out_AV_Transfer2 )
   END_RUNG wire#w1
   // the same network as SCL:
   #"AV-20.05"(LOCK := #"lock 1",   // "Valve"
               LIOP_SEL := #init,
               L_AUT := #init,
               L_REMOTE := #init,
               L_RESET := #reset,
               AUT_OP := "Blend_T-20".Out_AV_Transfer2,
               L_MON := #init,
               INSTANCE := 'AV-20.05',
               QCMD_OP => "AV-20.05");
END_REGION

REGION Network 8: AV-20.06 w ZSC
   RUNG wire#powerrail
      #"AV-20.06"(AUT_OP := wire#w1, LOCK := #"lock 1", ERR_EXTERN :=, LIOP_SEL := #init, L_AUT := #init, L_REMOTE := #init, L_SIM :=, L_RESET := #reset, MAN_OP :=, SIM_OP :=, FB_OPEN :=, FB_CLOSE :=, L_MON := #init, MON_T :=, MON_T_CLOSE :=, INSTANCE := 'AV-20.06', RESTART :=, VISIBILITY :=, OPdwCmd :=, QdwState =>, QwState =>, QCLOSING =>, QCLOSE =>, QOPENING =>, QOPEN =>, QCMD_OP => "AV-20.06", QMON =>, QMON_ERR =>, QMON_T =>, QMON_T_CLOSE =>, QMAN_AUT =>, QREMOTE =>, QSIM =>, QLOCK =>, QERR =>, QERR_EXT =>, QwAlarm =>)
   END_RUNG
   RUNG wire#powerrail
      Contact( "Blend_T-20".Out_AV_Transfer2 )
   END_RUNG wire#w1
   // the same network as SCL:
   #"AV-20.06"(LOCK := #"lock 1",   // "Valve"
               LIOP_SEL := #init,
               L_AUT := #init,
               L_REMOTE := #init,
               L_RESET := #reset,
               AUT_OP := "Blend_T-20".Out_AV_Transfer2,
               L_MON := #init,
               INSTANCE := 'AV-20.06',
               QCMD_OP => "AV-20.06");
END_REGION

REGION Network 9: AV-20.07
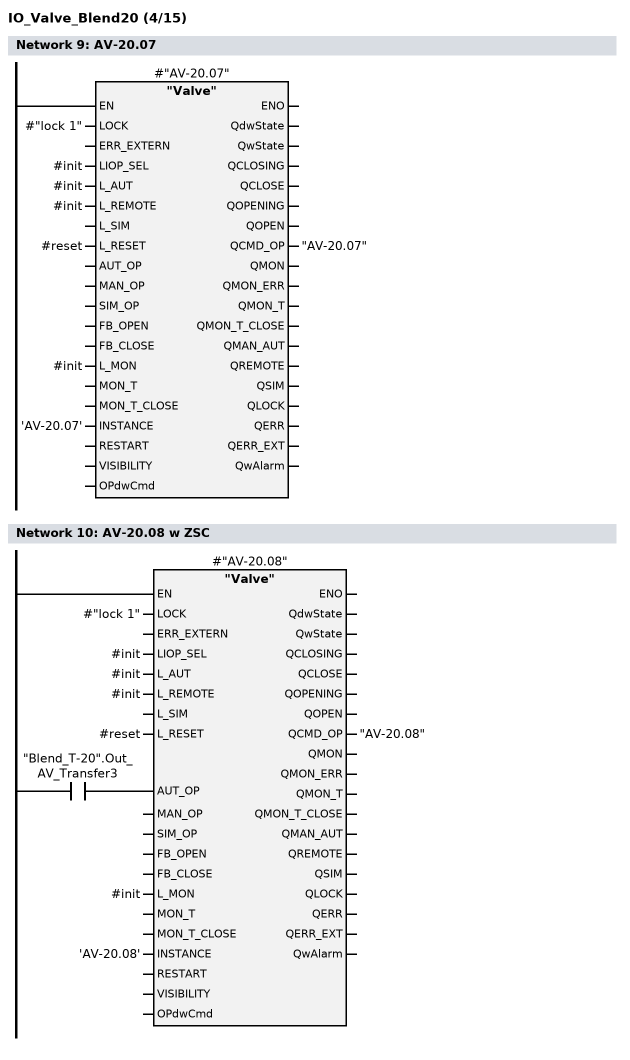
   RUNG wire#powerrail
      #"AV-20.07"(LOCK := #"lock 1", ERR_EXTERN :=, LIOP_SEL := #init, L_AUT := #init, L_REMOTE := #init, L_SIM :=, L_RESET := #reset, AUT_OP :=, MAN_OP :=, SIM_OP :=, FB_OPEN :=, FB_CLOSE :=, L_MON := #init, MON_T :=, MON_T_CLOSE :=, INSTANCE := 'AV-20.07', RESTART :=, VISIBILITY :=, OPdwCmd :=, QdwState =>, QwState =>, QCLOSING =>, QCLOSE =>, QOPENING =>, QOPEN =>, QCMD_OP => "AV-20.07", QMON =>, QMON_ERR =>, QMON_T =>, QMON_T_CLOSE =>, QMAN_AUT =>, QREMOTE =>, QSIM =>, QLOCK =>, QERR =>, QERR_EXT =>, QwAlarm =>)
   END_RUNG
   // the same network as SCL:
   #"AV-20.07"(LOCK := #"lock 1",   // "Valve"
               LIOP_SEL := #init,
               L_AUT := #init,
               L_REMOTE := #init,
               L_RESET := #reset,
               L_MON := #init,
               INSTANCE := 'AV-20.07',
               QCMD_OP => "AV-20.07");
END_REGION

REGION Network 10: AV-20.08 w ZSC
   RUNG wire#powerrail
      #"AV-20.08"(AUT_OP := wire#w1, LOCK := #"lock 1", ERR_EXTERN :=, LIOP_SEL := #init, L_AUT := #init, L_REMOTE := #init, L_SIM :=, L_RESET := #reset, MAN_OP :=, SIM_OP :=, FB_OPEN :=, FB_CLOSE :=, L_MON := #init, MON_T :=, MON_T_CLOSE :=, INSTANCE := 'AV-20.08', RESTART :=, VISIBILITY :=, OPdwCmd :=, QdwState =>, QwState =>, QCLOSING =>, QCLOSE =>, QOPENING =>, QOPEN =>, QCMD_OP => "AV-20.08", QMON =>, QMON_ERR =>, QMON_T =>, QMON_T_CLOSE =>, QMAN_AUT =>, QREMOTE =>, QSIM =>, QLOCK =>, QERR =>, QERR_EXT =>, QwAlarm =>)
   END_RUNG
   RUNG wire#powerrail
      Contact( "Blend_T-20".Out_AV_Transfer3 )
   END_RUNG wire#w1
   // the same network as SCL:
   #"AV-20.08"(LOCK := #"lock 1",   // "Valve"
               LIOP_SEL := #init,
               L_AUT := #init,
               L_REMOTE := #init,
               L_RESET := #reset,
               AUT_OP := "Blend_T-20".Out_AV_Transfer3,
               L_MON := #init,
               INSTANCE := 'AV-20.08',
               QCMD_OP => "AV-20.08");
END_REGION

REGION Network 11: AV-20.09 w ZSC
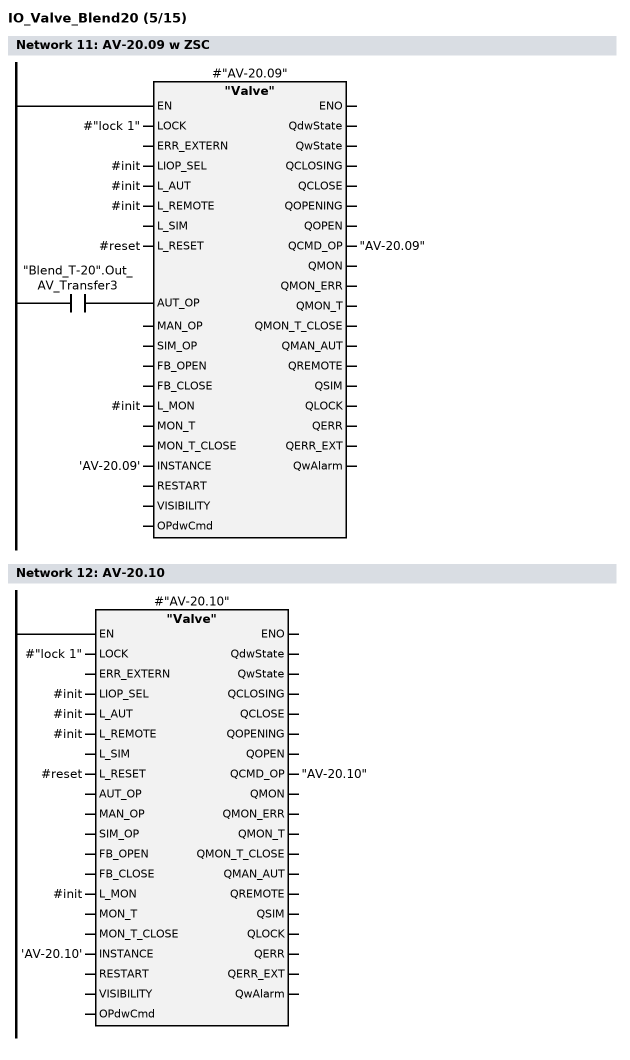
   RUNG wire#powerrail
      #"AV-20.09"(AUT_OP := wire#w1, LOCK := #"lock 1", ERR_EXTERN :=, LIOP_SEL := #init, L_AUT := #init, L_REMOTE := #init, L_SIM :=, L_RESET := #reset, MAN_OP :=, SIM_OP :=, FB_OPEN :=, FB_CLOSE :=, L_MON := #init, MON_T :=, MON_T_CLOSE :=, INSTANCE := 'AV-20.09', RESTART :=, VISIBILITY :=, OPdwCmd :=, QdwState =>, QwState =>, QCLOSING =>, QCLOSE =>, QOPENING =>, QOPEN =>, QCMD_OP => "AV-20.09", QMON =>, QMON_ERR =>, QMON_T =>, QMON_T_CLOSE =>, QMAN_AUT =>, QREMOTE =>, QSIM =>, QLOCK =>, QERR =>, QERR_EXT =>, QwAlarm =>)
   END_RUNG
   RUNG wire#powerrail
      Contact( "Blend_T-20".Out_AV_Transfer3 )
   END_RUNG wire#w1
   // the same network as SCL:
   #"AV-20.09"(LOCK := #"lock 1",   // "Valve"
               LIOP_SEL := #init,
               L_AUT := #init,
               L_REMOTE := #init,
               L_RESET := #reset,
               AUT_OP := "Blend_T-20".Out_AV_Transfer3,
               L_MON := #init,
               INSTANCE := 'AV-20.09',
               QCMD_OP => "AV-20.09");
END_REGION

REGION Network 12: AV-20.10
   RUNG wire#powerrail
      #"AV-20.10"(LOCK := #"lock 1", ERR_EXTERN :=, LIOP_SEL := #init, L_AUT := #init, L_REMOTE := #init, L_SIM :=, L_RESET := #reset, AUT_OP :=, MAN_OP :=, SIM_OP :=, FB_OPEN :=, FB_CLOSE :=, L_MON := #init, MON_T :=, MON_T_CLOSE :=, INSTANCE := 'AV-20.10', RESTART :=, VISIBILITY :=, OPdwCmd :=, QdwState =>, QwState =>, QCLOSING =>, QCLOSE =>, QOPENING =>, QOPEN =>, QCMD_OP => "AV-20.10", QMON =>, QMON_ERR =>, QMON_T =>, QMON_T_CLOSE =>, QMAN_AUT =>, QREMOTE =>, QSIM =>, QLOCK =>, QERR =>, QERR_EXT =>, QwAlarm =>)
   END_RUNG
   // the same network as SCL:
   #"AV-20.10"(LOCK := #"lock 1",   // "Valve"
               LIOP_SEL := #init,
               L_AUT := #init,
               L_REMOTE := #init,
               L_RESET := #reset,
               L_MON := #init,
               INSTANCE := 'AV-20.10',
               QCMD_OP => "AV-20.10");
END_REGION

REGION Network 13: AV-20.11 w ZSC
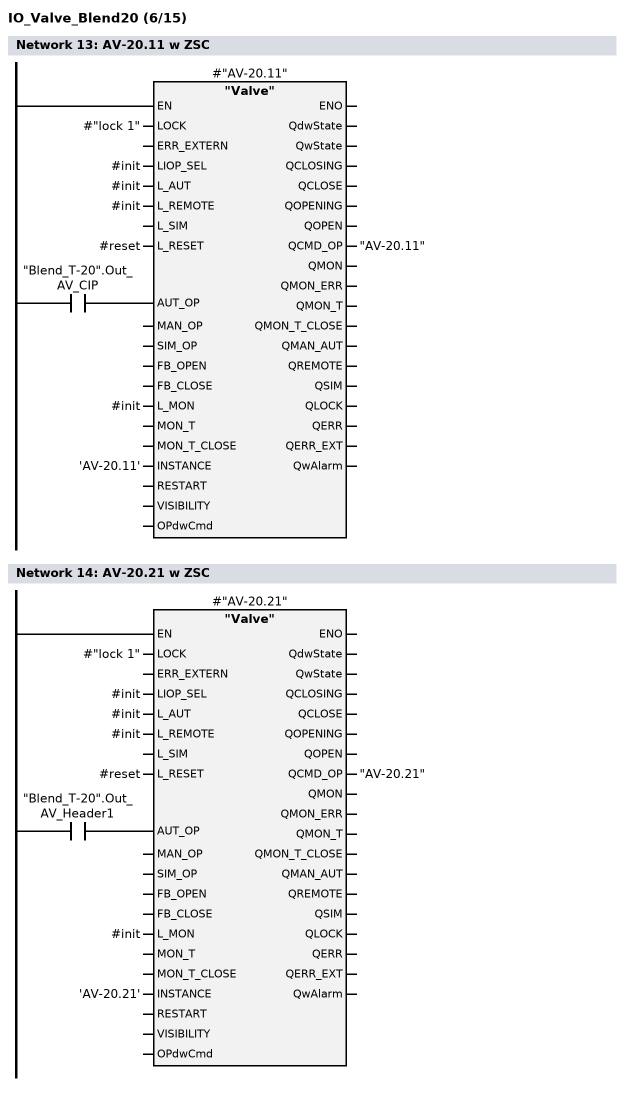
   RUNG wire#powerrail
      #"AV-20.11"(AUT_OP := wire#w1, LOCK := #"lock 1", ERR_EXTERN :=, LIOP_SEL := #init, L_AUT := #init, L_REMOTE := #init, L_SIM :=, L_RESET := #reset, MAN_OP :=, SIM_OP :=, FB_OPEN :=, FB_CLOSE :=, L_MON := #init, MON_T :=, MON_T_CLOSE :=, INSTANCE := 'AV-20.11', RESTART :=, VISIBILITY :=, OPdwCmd :=, QdwState =>, QwState =>, QCLOSING =>, QCLOSE =>, QOPENING =>, QOPEN =>, QCMD_OP => "AV-20.11", QMON =>, QMON_ERR =>, QMON_T =>, QMON_T_CLOSE =>, QMAN_AUT =>, QREMOTE =>, QSIM =>, QLOCK =>, QERR =>, QERR_EXT =>, QwAlarm =>)
   END_RUNG
   RUNG wire#powerrail
      Contact( "Blend_T-20".Out_AV_CIP )
   END_RUNG wire#w1
   // the same network as SCL:
   #"AV-20.11"(LOCK := #"lock 1",   // "Valve"
               LIOP_SEL := #init,
               L_AUT := #init,
               L_REMOTE := #init,
               L_RESET := #reset,
               AUT_OP := "Blend_T-20".Out_AV_CIP,
               L_MON := #init,
               INSTANCE := 'AV-20.11',
               QCMD_OP => "AV-20.11");
END_REGION

REGION Network 14: AV-20.21 w ZSC
   RUNG wire#powerrail
      #"AV-20.21"(AUT_OP := wire#w1, LOCK := #"lock 1", ERR_EXTERN :=, LIOP_SEL := #init, L_AUT := #init, L_REMOTE := #init, L_SIM :=, L_RESET := #reset, MAN_OP :=, SIM_OP :=, FB_OPEN :=, FB_CLOSE :=, L_MON := #init, MON_T :=, MON_T_CLOSE :=, INSTANCE := 'AV-20.21', RESTART :=, VISIBILITY :=, OPdwCmd :=, QdwState =>, QwState =>, QCLOSING =>, QCLOSE =>, QOPENING =>, QOPEN =>, QCMD_OP => "AV-20.21", QMON =>, QMON_ERR =>, QMON_T =>, QMON_T_CLOSE =>, QMAN_AUT =>, QREMOTE =>, QSIM =>, QLOCK =>, QERR =>, QERR_EXT =>, QwAlarm =>)
   END_RUNG
   RUNG wire#powerrail
      Contact( "Blend_T-20".Out_AV_Header1 )
   END_RUNG wire#w1
   // the same network as SCL:
   #"AV-20.21"(LOCK := #"lock 1",   // "Valve"
               LIOP_SEL := #init,
               L_AUT := #init,
               L_REMOTE := #init,
               L_RESET := #reset,
               AUT_OP := "Blend_T-20".Out_AV_Header1,
               L_MON := #init,
               INSTANCE := 'AV-20.21',
               QCMD_OP => "AV-20.21");
END_REGION

REGION Network 15: AV-20.22
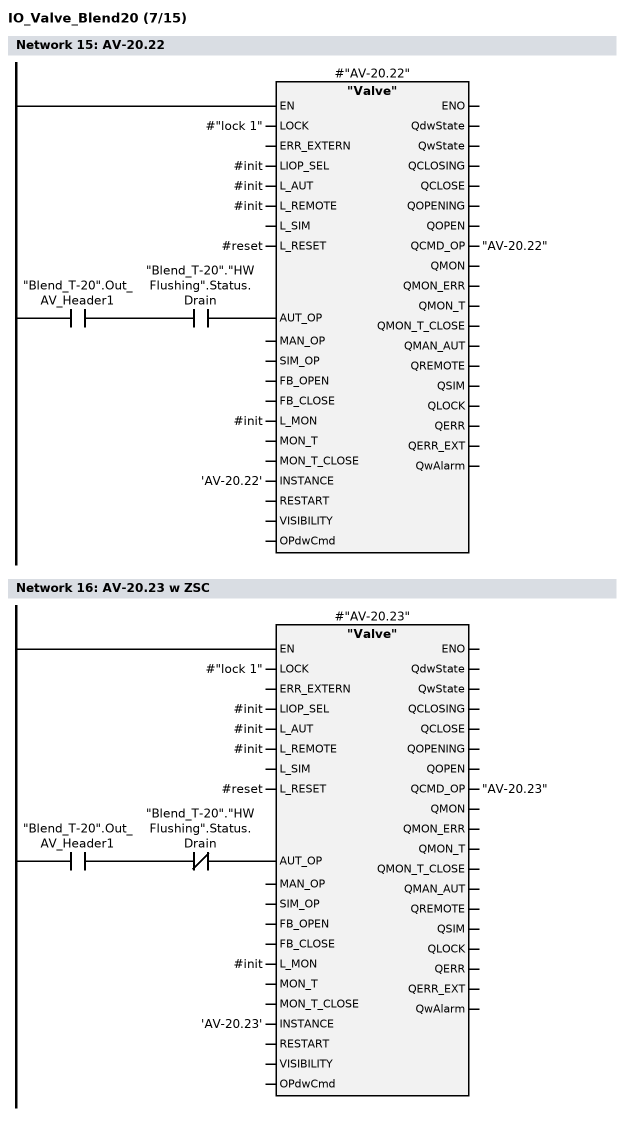
   RUNG wire#powerrail
      #"AV-20.22"(AUT_OP := wire#w1, LOCK := #"lock 1", ERR_EXTERN :=, LIOP_SEL := #init, L_AUT := #init, L_REMOTE := #init, L_SIM :=, L_RESET := #reset, MAN_OP :=, SIM_OP :=, FB_OPEN :=, FB_CLOSE :=, L_MON := #init, MON_T :=, MON_T_CLOSE :=, INSTANCE := 'AV-20.22', RESTART :=, VISIBILITY :=, OPdwCmd :=, QdwState =>, QwState =>, QCLOSING =>, QCLOSE =>, QOPENING =>, QOPEN =>, QCMD_OP => "AV-20.22", QMON =>, QMON_ERR =>, QMON_T =>, QMON_T_CLOSE =>, QMAN_AUT =>, QREMOTE =>, QSIM =>, QLOCK =>, QERR =>, QERR_EXT =>, QwAlarm =>)
   END_RUNG
   RUNG wire#powerrail
      Contact( "Blend_T-20".Out_AV_Header1 )
      Contact( "Blend_T-20"."HW Flushing".Status.Drain )
   END_RUNG wire#w1
   // the same network as SCL:
   #"AV-20.22"(LOCK := #"lock 1",   // "Valve"
               LIOP_SEL := #init,
               L_AUT := #init,
               L_REMOTE := #init,
               L_RESET := #reset,
               AUT_OP := "Blend_T-20".Out_AV_Header1 AND "Blend_T-20"."HW Flushing".Status.Drain,
               L_MON := #init,
               INSTANCE := 'AV-20.22',
               QCMD_OP => "AV-20.22");
END_REGION

REGION Network 16: AV-20.23 w ZSC
   RUNG wire#powerrail
      #"AV-20.23"(AUT_OP := wire#w1, LOCK := #"lock 1", ERR_EXTERN :=, LIOP_SEL := #init, L_AUT := #init, L_REMOTE := #init, L_SIM :=, L_RESET := #reset, MAN_OP :=, SIM_OP :=, FB_OPEN :=, FB_CLOSE :=, L_MON := #init, MON_T :=, MON_T_CLOSE :=, INSTANCE := 'AV-20.23', RESTART :=, VISIBILITY :=, OPdwCmd :=, QdwState =>, QwState =>, QCLOSING =>, QCLOSE =>, QOPENING =>, QOPEN =>, QCMD_OP => "AV-20.23", QMON =>, QMON_ERR =>, QMON_T =>, QMON_T_CLOSE =>, QMAN_AUT =>, QREMOTE =>, QSIM =>, QLOCK =>, QERR =>, QERR_EXT =>, QwAlarm =>)
   END_RUNG
   RUNG wire#powerrail
      Contact( "Blend_T-20".Out_AV_Header1 )
      I_Contact( "Blend_T-20"."HW Flushing".Status.Drain )
   END_RUNG wire#w1
   // the same network as SCL:
   #"AV-20.23"(LOCK := #"lock 1",   // "Valve"
               LIOP_SEL := #init,
               L_AUT := #init,
               L_REMOTE := #init,
               L_RESET := #reset,
               AUT_OP := "Blend_T-20".Out_AV_Header1 AND NOT "Blend_T-20"."HW Flushing".Status.Drain,
               L_MON := #init,
               INSTANCE := 'AV-20.23',
               QCMD_OP => "AV-20.23");
END_REGION

REGION Network 17: AV-20.24 w ZSC
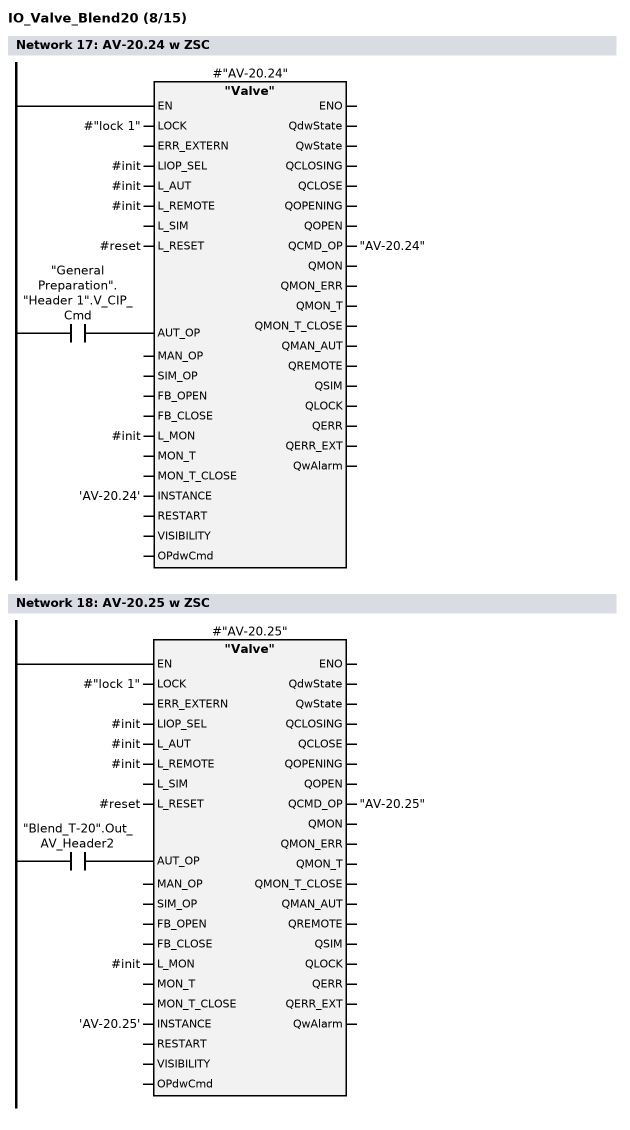
   RUNG wire#powerrail
      #"AV-20.24"(AUT_OP := wire#w1, LOCK := #"lock 1", ERR_EXTERN :=, LIOP_SEL := #init, L_AUT := #init, L_REMOTE := #init, L_SIM :=, L_RESET := #reset, MAN_OP :=, SIM_OP :=, FB_OPEN :=, FB_CLOSE :=, L_MON := #init, MON_T :=, MON_T_CLOSE :=, INSTANCE := 'AV-20.24', RESTART :=, VISIBILITY :=, OPdwCmd :=, QdwState =>, QwState =>, QCLOSING =>, QCLOSE =>, QOPENING =>, QOPEN =>, QCMD_OP => "AV-20.24", QMON =>, QMON_ERR =>, QMON_T =>, QMON_T_CLOSE =>, QMAN_AUT =>, QREMOTE =>, QSIM =>, QLOCK =>, QERR =>, QERR_EXT =>, QwAlarm =>)
   END_RUNG
   RUNG wire#powerrail
      Contact( "General Preparation"."Header 1".V_CIP_Cmd )
   END_RUNG wire#w1
   // the same network as SCL:
   #"AV-20.24"(LOCK := #"lock 1",   // "Valve"
               LIOP_SEL := #init,
               L_AUT := #init,
               L_REMOTE := #init,
               L_RESET := #reset,
               AUT_OP := "General Preparation"."Header 1".V_CIP_Cmd,
               L_MON := #init,
               INSTANCE := 'AV-20.24',
               QCMD_OP => "AV-20.24");
END_REGION

REGION Network 18: AV-20.25 w ZSC
   RUNG wire#powerrail
      #"AV-20.25"(AUT_OP := wire#w1, LOCK := #"lock 1", ERR_EXTERN :=, LIOP_SEL := #init, L_AUT := #init, L_REMOTE := #init, L_SIM :=, L_RESET := #reset, MAN_OP :=, SIM_OP :=, FB_OPEN :=, FB_CLOSE :=, L_MON := #init, MON_T :=, MON_T_CLOSE :=, INSTANCE := 'AV-20.25', RESTART :=, VISIBILITY :=, OPdwCmd :=, QdwState =>, QwState =>, QCLOSING =>, QCLOSE =>, QOPENING =>, QOPEN =>, QCMD_OP => "AV-20.25", QMON =>, QMON_ERR =>, QMON_T =>, QMON_T_CLOSE =>, QMAN_AUT =>, QREMOTE =>, QSIM =>, QLOCK =>, QERR =>, QERR_EXT =>, QwAlarm =>)
   END_RUNG
   RUNG wire#powerrail
      Contact( "Blend_T-20".Out_AV_Header2 )
   END_RUNG wire#w1
   // the same network as SCL:
   #"AV-20.25"(LOCK := #"lock 1",   // "Valve"
               LIOP_SEL := #init,
               L_AUT := #init,
               L_REMOTE := #init,
               L_RESET := #reset,
               AUT_OP := "Blend_T-20".Out_AV_Header2,
               L_MON := #init,
               INSTANCE := 'AV-20.25',
               QCMD_OP => "AV-20.25");
END_REGION

REGION Network 19: AV-20.26
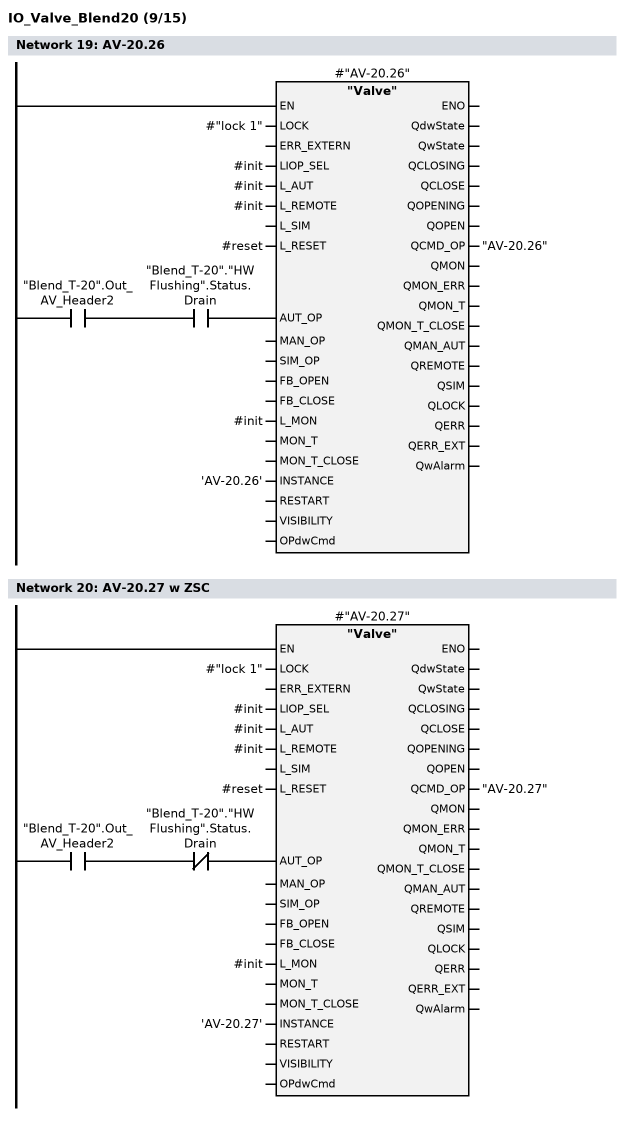
   RUNG wire#powerrail
      #"AV-20.26"(AUT_OP := wire#w1, LOCK := #"lock 1", ERR_EXTERN :=, LIOP_SEL := #init, L_AUT := #init, L_REMOTE := #init, L_SIM :=, L_RESET := #reset, MAN_OP :=, SIM_OP :=, FB_OPEN :=, FB_CLOSE :=, L_MON := #init, MON_T :=, MON_T_CLOSE :=, INSTANCE := 'AV-20.26', RESTART :=, VISIBILITY :=, OPdwCmd :=, QdwState =>, QwState =>, QCLOSING =>, QCLOSE =>, QOPENING =>, QOPEN =>, QCMD_OP => "AV-20.26", QMON =>, QMON_ERR =>, QMON_T =>, QMON_T_CLOSE =>, QMAN_AUT =>, QREMOTE =>, QSIM =>, QLOCK =>, QERR =>, QERR_EXT =>, QwAlarm =>)
   END_RUNG
   RUNG wire#powerrail
      Contact( "Blend_T-20".Out_AV_Header2 )
      Contact( "Blend_T-20"."HW Flushing".Status.Drain )
   END_RUNG wire#w1
   // the same network as SCL:
   #"AV-20.26"(LOCK := #"lock 1",   // "Valve"
               LIOP_SEL := #init,
               L_AUT := #init,
               L_REMOTE := #init,
               L_RESET := #reset,
               AUT_OP := "Blend_T-20".Out_AV_Header2 AND "Blend_T-20"."HW Flushing".Status.Drain,
               L_MON := #init,
               INSTANCE := 'AV-20.26',
               QCMD_OP => "AV-20.26");
END_REGION

REGION Network 20: AV-20.27 w ZSC
   RUNG wire#powerrail
      #"AV-20.27"(AUT_OP := wire#w1, LOCK := #"lock 1", ERR_EXTERN :=, LIOP_SEL := #init, L_AUT := #init, L_REMOTE := #init, L_SIM :=, L_RESET := #reset, MAN_OP :=, SIM_OP :=, FB_OPEN :=, FB_CLOSE :=, L_MON := #init, MON_T :=, MON_T_CLOSE :=, INSTANCE := 'AV-20.27', RESTART :=, VISIBILITY :=, OPdwCmd :=, QdwState =>, QwState =>, QCLOSING =>, QCLOSE =>, QOPENING =>, QOPEN =>, QCMD_OP => "AV-20.27", QMON =>, QMON_ERR =>, QMON_T =>, QMON_T_CLOSE =>, QMAN_AUT =>, QREMOTE =>, QSIM =>, QLOCK =>, QERR =>, QERR_EXT =>, QwAlarm =>)
   END_RUNG
   RUNG wire#powerrail
      Contact( "Blend_T-20".Out_AV_Header2 )
      I_Contact( "Blend_T-20"."HW Flushing".Status.Drain )
   END_RUNG wire#w1
   // the same network as SCL:
   #"AV-20.27"(LOCK := #"lock 1",   // "Valve"
               LIOP_SEL := #init,
               L_AUT := #init,
               L_REMOTE := #init,
               L_RESET := #reset,
               AUT_OP := "Blend_T-20".Out_AV_Header2 AND NOT "Blend_T-20"."HW Flushing".Status.Drain,
               L_MON := #init,
               INSTANCE := 'AV-20.27',
               QCMD_OP => "AV-20.27");
END_REGION

REGION Network 21: AV-20.28 w ZSC
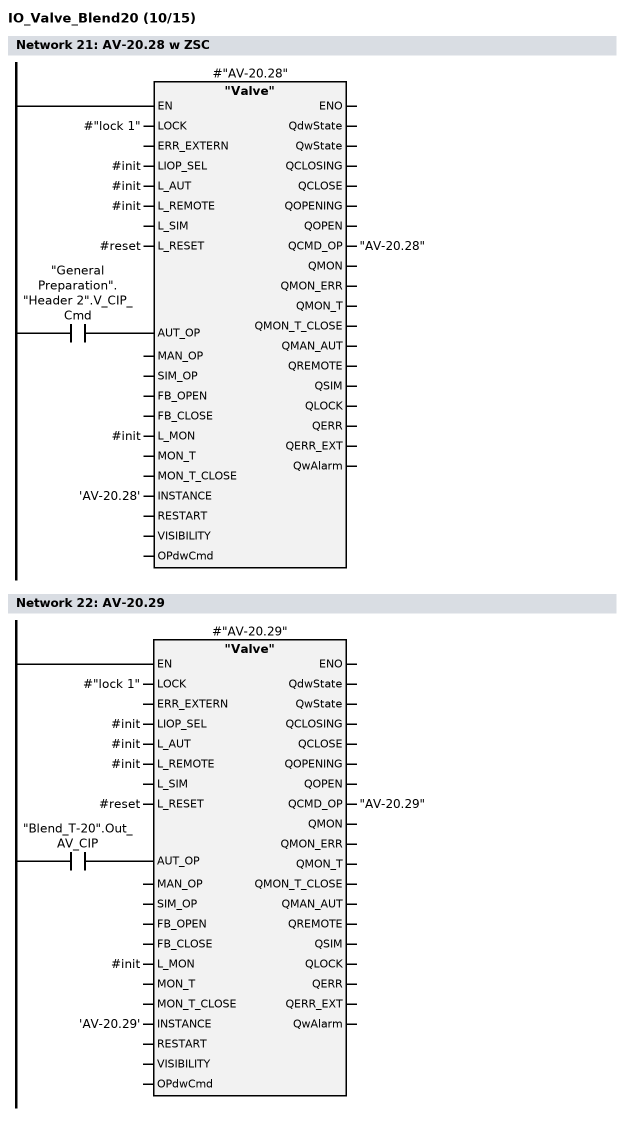
   RUNG wire#powerrail
      #"AV-20.28"(AUT_OP := wire#w1, LOCK := #"lock 1", ERR_EXTERN :=, LIOP_SEL := #init, L_AUT := #init, L_REMOTE := #init, L_SIM :=, L_RESET := #reset, MAN_OP :=, SIM_OP :=, FB_OPEN :=, FB_CLOSE :=, L_MON := #init, MON_T :=, MON_T_CLOSE :=, INSTANCE := 'AV-20.28', RESTART :=, VISIBILITY :=, OPdwCmd :=, QdwState =>, QwState =>, QCLOSING =>, QCLOSE =>, QOPENING =>, QOPEN =>, QCMD_OP => "AV-20.28", QMON =>, QMON_ERR =>, QMON_T =>, QMON_T_CLOSE =>, QMAN_AUT =>, QREMOTE =>, QSIM =>, QLOCK =>, QERR =>, QERR_EXT =>, QwAlarm =>)
   END_RUNG
   RUNG wire#powerrail
      Contact( "General Preparation"."Header 2".V_CIP_Cmd )
   END_RUNG wire#w1
   // the same network as SCL:
   #"AV-20.28"(LOCK := #"lock 1",   // "Valve"
               LIOP_SEL := #init,
               L_AUT := #init,
               L_REMOTE := #init,
               L_RESET := #reset,
               AUT_OP := "General Preparation"."Header 2".V_CIP_Cmd,
               L_MON := #init,
               INSTANCE := 'AV-20.28',
               QCMD_OP => "AV-20.28");
END_REGION

REGION Network 22: AV-20.29
   RUNG wire#powerrail
      #"AV-20.29"(AUT_OP := wire#w1, LOCK := #"lock 1", ERR_EXTERN :=, LIOP_SEL := #init, L_AUT := #init, L_REMOTE := #init, L_SIM :=, L_RESET := #reset, MAN_OP :=, SIM_OP :=, FB_OPEN :=, FB_CLOSE :=, L_MON := #init, MON_T :=, MON_T_CLOSE :=, INSTANCE := 'AV-20.29', RESTART :=, VISIBILITY :=, OPdwCmd :=, QdwState =>, QwState =>, QCLOSING =>, QCLOSE =>, QOPENING =>, QOPEN =>, QCMD_OP => "AV-20.29", QMON =>, QMON_ERR =>, QMON_T =>, QMON_T_CLOSE =>, QMAN_AUT =>, QREMOTE =>, QSIM =>, QLOCK =>, QERR =>, QERR_EXT =>, QwAlarm =>)
   END_RUNG
   RUNG wire#powerrail
      Contact( "Blend_T-20".Out_AV_CIP )
   END_RUNG wire#w1
   // the same network as SCL:
   #"AV-20.29"(LOCK := #"lock 1",   // "Valve"
               LIOP_SEL := #init,
               L_AUT := #init,
               L_REMOTE := #init,
               L_RESET := #reset,
               AUT_OP := "Blend_T-20".Out_AV_CIP,
               L_MON := #init,
               INSTANCE := 'AV-20.29',
               QCMD_OP => "AV-20.29");
END_REGION

REGION Network 23: AV-20.30
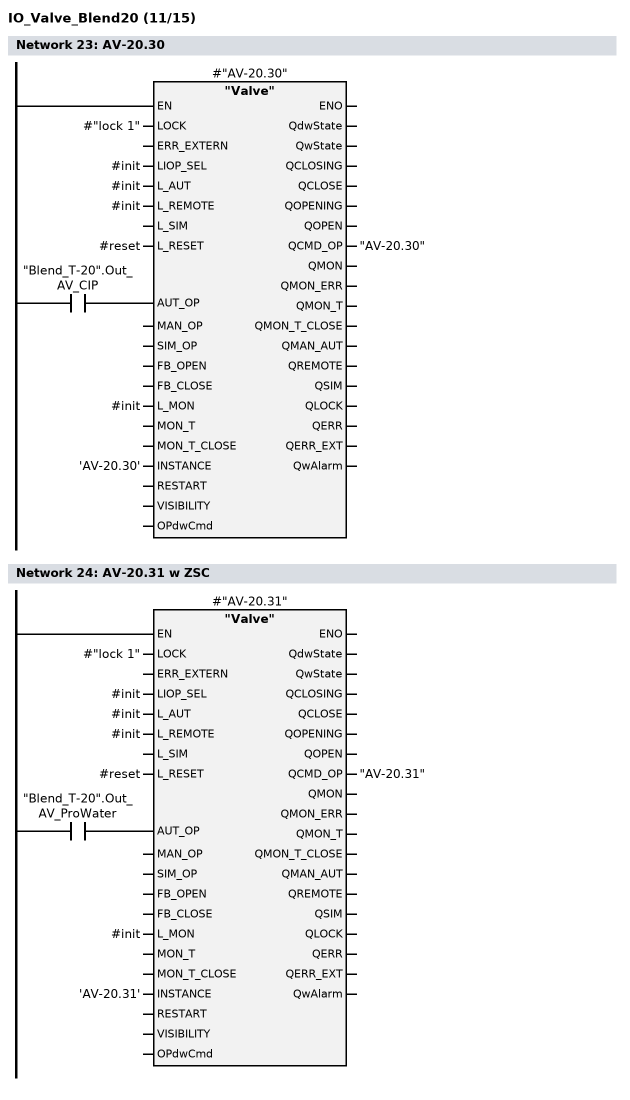
   RUNG wire#powerrail
      #"AV-20.30"(AUT_OP := wire#w1, LOCK := #"lock 1", ERR_EXTERN :=, LIOP_SEL := #init, L_AUT := #init, L_REMOTE := #init, L_SIM :=, L_RESET := #reset, MAN_OP :=, SIM_OP :=, FB_OPEN :=, FB_CLOSE :=, L_MON := #init, MON_T :=, MON_T_CLOSE :=, INSTANCE := 'AV-20.30', RESTART :=, VISIBILITY :=, OPdwCmd :=, QdwState =>, QwState =>, QCLOSING =>, QCLOSE =>, QOPENING =>, QOPEN =>, QCMD_OP => "AV-20.30", QMON =>, QMON_ERR =>, QMON_T =>, QMON_T_CLOSE =>, QMAN_AUT =>, QREMOTE =>, QSIM =>, QLOCK =>, QERR =>, QERR_EXT =>, QwAlarm =>)
   END_RUNG
   RUNG wire#powerrail
      Contact( "Blend_T-20".Out_AV_CIP )
   END_RUNG wire#w1
   // the same network as SCL:
   #"AV-20.30"(LOCK := #"lock 1",   // "Valve"
               LIOP_SEL := #init,
               L_AUT := #init,
               L_REMOTE := #init,
               L_RESET := #reset,
               AUT_OP := "Blend_T-20".Out_AV_CIP,
               L_MON := #init,
               INSTANCE := 'AV-20.30',
               QCMD_OP => "AV-20.30");
END_REGION

REGION Network 24: AV-20.31 w ZSC
   RUNG wire#powerrail
      #"AV-20.31"(AUT_OP := wire#w1, LOCK := #"lock 1", ERR_EXTERN :=, LIOP_SEL := #init, L_AUT := #init, L_REMOTE := #init, L_SIM :=, L_RESET := #reset, MAN_OP :=, SIM_OP :=, FB_OPEN :=, FB_CLOSE :=, L_MON := #init, MON_T :=, MON_T_CLOSE :=, INSTANCE := 'AV-20.31', RESTART :=, VISIBILITY :=, OPdwCmd :=, QdwState =>, QwState =>, QCLOSING =>, QCLOSE =>, QOPENING =>, QOPEN =>, QCMD_OP => "AV-20.31", QMON =>, QMON_ERR =>, QMON_T =>, QMON_T_CLOSE =>, QMAN_AUT =>, QREMOTE =>, QSIM =>, QLOCK =>, QERR =>, QERR_EXT =>, QwAlarm =>)
   END_RUNG
   RUNG wire#powerrail
      Contact( "Blend_T-20".Out_AV_ProWater )
   END_RUNG wire#w1
   // the same network as SCL:
   #"AV-20.31"(LOCK := #"lock 1",   // "Valve"
               LIOP_SEL := #init,
               L_AUT := #init,
               L_REMOTE := #init,
               L_RESET := #reset,
               AUT_OP := "Blend_T-20".Out_AV_ProWater,
               L_MON := #init,
               INSTANCE := 'AV-20.31',
               QCMD_OP => "AV-20.31");
END_REGION

REGION Network 25: AV-20.32 w ZSC
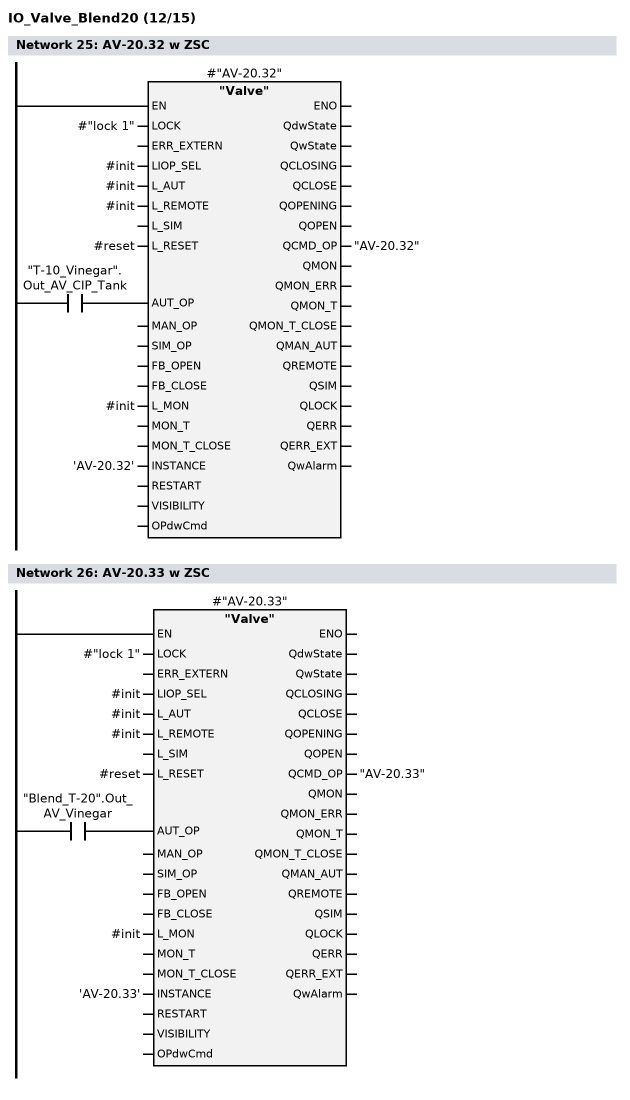
   RUNG wire#powerrail
      #"AV-20.32"(AUT_OP := wire#w1, LOCK := #"lock 1", ERR_EXTERN :=, LIOP_SEL := #init, L_AUT := #init, L_REMOTE := #init, L_SIM :=, L_RESET := #reset, MAN_OP :=, SIM_OP :=, FB_OPEN :=, FB_CLOSE :=, L_MON := #init, MON_T :=, MON_T_CLOSE :=, INSTANCE := 'AV-20.32', RESTART :=, VISIBILITY :=, OPdwCmd :=, QdwState =>, QwState =>, QCLOSING =>, QCLOSE =>, QOPENING =>, QOPEN =>, QCMD_OP => "AV-20.32", QMON =>, QMON_ERR =>, QMON_T =>, QMON_T_CLOSE =>, QMAN_AUT =>, QREMOTE =>, QSIM =>, QLOCK =>, QERR =>, QERR_EXT =>, QwAlarm =>)
   END_RUNG
   RUNG wire#powerrail
      Contact( "T-10_Vinegar".Out_AV_CIP_Tank )
   END_RUNG wire#w1
   // the same network as SCL:
   #"AV-20.32"(LOCK := #"lock 1",   // "Valve"
               LIOP_SEL := #init,
               L_AUT := #init,
               L_REMOTE := #init,
               L_RESET := #reset,
               AUT_OP := "T-10_Vinegar".Out_AV_CIP_Tank,
               L_MON := #init,
               INSTANCE := 'AV-20.32',
               QCMD_OP => "AV-20.32");
END_REGION

REGION Network 26: AV-20.33 w ZSC
   RUNG wire#powerrail
      #"AV-20.33"(AUT_OP := wire#w1, LOCK := #"lock 1", ERR_EXTERN :=, LIOP_SEL := #init, L_AUT := #init, L_REMOTE := #init, L_SIM :=, L_RESET := #reset, MAN_OP :=, SIM_OP :=, FB_OPEN :=, FB_CLOSE :=, L_MON := #init, MON_T :=, MON_T_CLOSE :=, INSTANCE := 'AV-20.33', RESTART :=, VISIBILITY :=, OPdwCmd :=, QdwState =>, QwState =>, QCLOSING =>, QCLOSE =>, QOPENING =>, QOPEN =>, QCMD_OP => "AV-20.33", QMON =>, QMON_ERR =>, QMON_T =>, QMON_T_CLOSE =>, QMAN_AUT =>, QREMOTE =>, QSIM =>, QLOCK =>, QERR =>, QERR_EXT =>, QwAlarm =>)
   END_RUNG
   RUNG wire#powerrail
      Contact( "Blend_T-20".Out_AV_Vinegar )
   END_RUNG wire#w1
   // the same network as SCL:
   #"AV-20.33"(LOCK := #"lock 1",   // "Valve"
               LIOP_SEL := #init,
               L_AUT := #init,
               L_REMOTE := #init,
               L_RESET := #reset,
               AUT_OP := "Blend_T-20".Out_AV_Vinegar,
               L_MON := #init,
               INSTANCE := 'AV-20.33',
               QCMD_OP => "AV-20.33");
END_REGION

REGION Network 27: AV-20.34 w ZSC
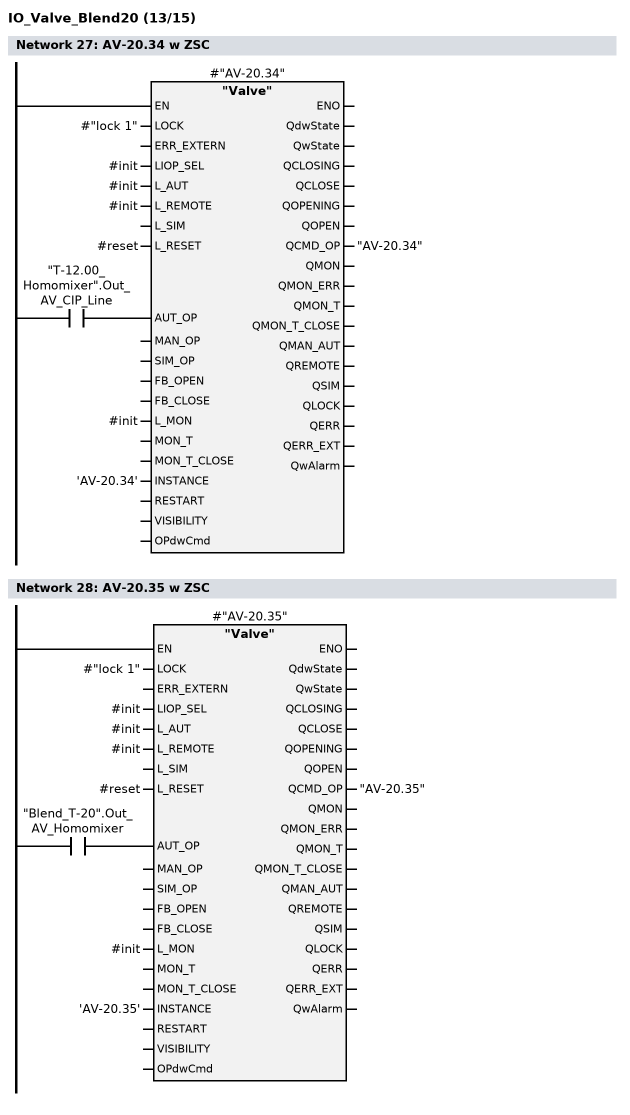
   RUNG wire#powerrail
      #"AV-20.34"(AUT_OP := wire#w1, LOCK := #"lock 1", ERR_EXTERN :=, LIOP_SEL := #init, L_AUT := #init, L_REMOTE := #init, L_SIM :=, L_RESET := #reset, MAN_OP :=, SIM_OP :=, FB_OPEN :=, FB_CLOSE :=, L_MON := #init, MON_T :=, MON_T_CLOSE :=, INSTANCE := 'AV-20.34', RESTART :=, VISIBILITY :=, OPdwCmd :=, QdwState =>, QwState =>, QCLOSING =>, QCLOSE =>, QOPENING =>, QOPEN =>, QCMD_OP => "AV-20.34", QMON =>, QMON_ERR =>, QMON_T =>, QMON_T_CLOSE =>, QMAN_AUT =>, QREMOTE =>, QSIM =>, QLOCK =>, QERR =>, QERR_EXT =>, QwAlarm =>)
   END_RUNG
   RUNG wire#powerrail
      Contact( "T-12.00_Homomixer".Out_AV_CIP_Line )
   END_RUNG wire#w1
   // the same network as SCL:
   #"AV-20.34"(LOCK := #"lock 1",   // "Valve"
               LIOP_SEL := #init,
               L_AUT := #init,
               L_REMOTE := #init,
               L_RESET := #reset,
               AUT_OP := "T-12.00_Homomixer".Out_AV_CIP_Line,
               L_MON := #init,
               INSTANCE := 'AV-20.34',
               QCMD_OP => "AV-20.34");
END_REGION

REGION Network 28: AV-20.35 w ZSC
   RUNG wire#powerrail
      #"AV-20.35"(AUT_OP := wire#w1, LOCK := #"lock 1", ERR_EXTERN :=, LIOP_SEL := #init, L_AUT := #init, L_REMOTE := #init, L_SIM :=, L_RESET := #reset, MAN_OP :=, SIM_OP :=, FB_OPEN :=, FB_CLOSE :=, L_MON := #init, MON_T :=, MON_T_CLOSE :=, INSTANCE := 'AV-20.35', RESTART :=, VISIBILITY :=, OPdwCmd :=, QdwState =>, QwState =>, QCLOSING =>, QCLOSE =>, QOPENING =>, QOPEN =>, QCMD_OP => "AV-20.35", QMON =>, QMON_ERR =>, QMON_T =>, QMON_T_CLOSE =>, QMAN_AUT =>, QREMOTE =>, QSIM =>, QLOCK =>, QERR =>, QERR_EXT =>, QwAlarm =>)
   END_RUNG
   RUNG wire#powerrail
      Contact( "Blend_T-20".Out_AV_Homomixer )
   END_RUNG wire#w1
   // the same network as SCL:
   #"AV-20.35"(LOCK := #"lock 1",   // "Valve"
               LIOP_SEL := #init,
               L_AUT := #init,
               L_REMOTE := #init,
               L_RESET := #reset,
               AUT_OP := "Blend_T-20".Out_AV_Homomixer,
               L_MON := #init,
               INSTANCE := 'AV-20.35',
               QCMD_OP => "AV-20.35");
END_REGION

REGION Network 29: AV-20.36 w ZSC
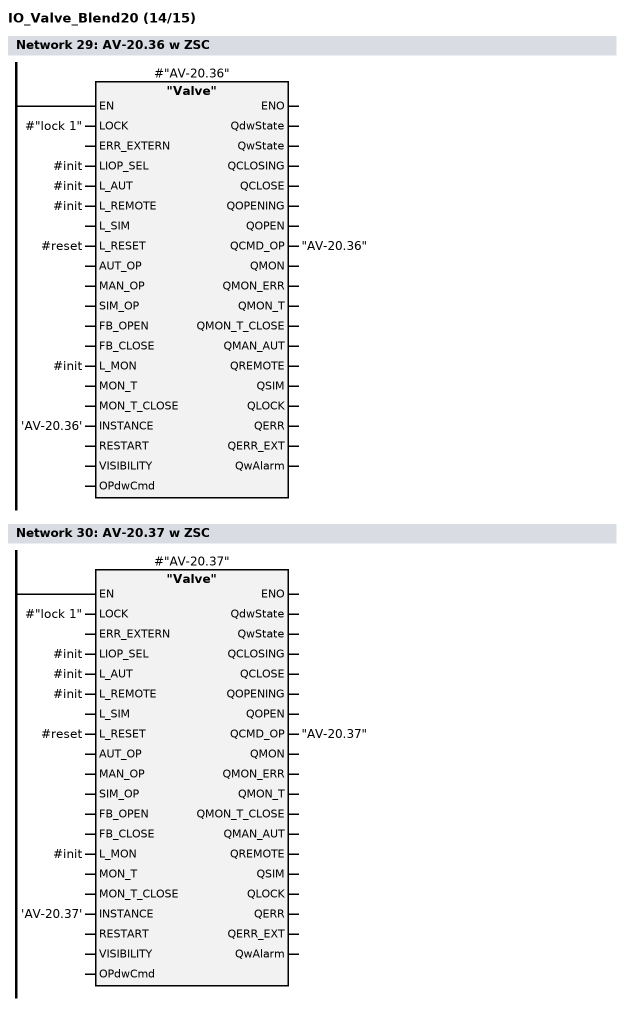
   RUNG wire#powerrail
      #"AV-20.36"(LOCK := #"lock 1", ERR_EXTERN :=, LIOP_SEL := #init, L_AUT := #init, L_REMOTE := #init, L_SIM :=, L_RESET := #reset, AUT_OP :=, MAN_OP :=, SIM_OP :=, FB_OPEN :=, FB_CLOSE :=, L_MON := #init, MON_T :=, MON_T_CLOSE :=, INSTANCE := 'AV-20.36', RESTART :=, VISIBILITY :=, OPdwCmd :=, QdwState =>, QwState =>, QCLOSING =>, QCLOSE =>, QOPENING =>, QOPEN =>, QCMD_OP => "AV-20.36", QMON =>, QMON_ERR =>, QMON_T =>, QMON_T_CLOSE =>, QMAN_AUT =>, QREMOTE =>, QSIM =>, QLOCK =>, QERR =>, QERR_EXT =>, QwAlarm =>)
   END_RUNG
   // the same network as SCL:
   #"AV-20.36"(LOCK := #"lock 1",   // "Valve"
               LIOP_SEL := #init,
               L_AUT := #init,
               L_REMOTE := #init,
               L_RESET := #reset,
               L_MON := #init,
               INSTANCE := 'AV-20.36',
               QCMD_OP => "AV-20.36");
END_REGION

REGION Network 30: AV-20.37 w ZSC
   RUNG wire#powerrail
      #"AV-20.37"(LOCK := #"lock 1", ERR_EXTERN :=, LIOP_SEL := #init, L_AUT := #init, L_REMOTE := #init, L_SIM :=, L_RESET := #reset, AUT_OP :=, MAN_OP :=, SIM_OP :=, FB_OPEN :=, FB_CLOSE :=, L_MON := #init, MON_T :=, MON_T_CLOSE :=, INSTANCE := 'AV-20.37', RESTART :=, VISIBILITY :=, OPdwCmd :=, QdwState =>, QwState =>, QCLOSING =>, QCLOSE =>, QOPENING =>, QOPEN =>, QCMD_OP => "AV-20.37", QMON =>, QMON_ERR =>, QMON_T =>, QMON_T_CLOSE =>, QMAN_AUT =>, QREMOTE =>, QSIM =>, QLOCK =>, QERR =>, QERR_EXT =>, QwAlarm =>)
   END_RUNG
   // the same network as SCL:
   #"AV-20.37"(LOCK := #"lock 1",   // "Valve"
               LIOP_SEL := #init,
               L_AUT := #init,
               L_REMOTE := #init,
               L_RESET := #reset,
               L_MON := #init,
               INSTANCE := 'AV-20.37',
               QCMD_OP => "AV-20.37");
END_REGION

REGION Network 31: AV-20.41
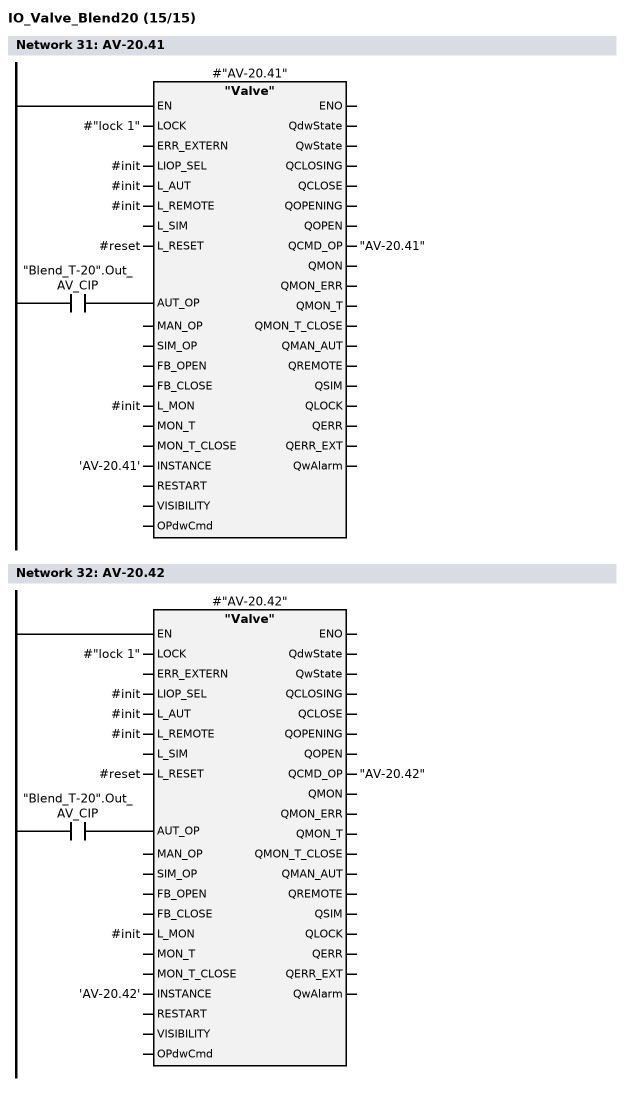
   RUNG wire#powerrail
      #"AV-20.41"(AUT_OP := wire#w1, LOCK := #"lock 1", ERR_EXTERN :=, LIOP_SEL := #init, L_AUT := #init, L_REMOTE := #init, L_SIM :=, L_RESET := #reset, MAN_OP :=, SIM_OP :=, FB_OPEN :=, FB_CLOSE :=, L_MON := #init, MON_T :=, MON_T_CLOSE :=, INSTANCE := 'AV-20.41', RESTART :=, VISIBILITY :=, OPdwCmd :=, QdwState =>, QwState =>, QCLOSING =>, QCLOSE =>, QOPENING =>, QOPEN =>, QCMD_OP => "AV-20.41", QMON =>, QMON_ERR =>, QMON_T =>, QMON_T_CLOSE =>, QMAN_AUT =>, QREMOTE =>, QSIM =>, QLOCK =>, QERR =>, QERR_EXT =>, QwAlarm =>)
   END_RUNG
   RUNG wire#powerrail
      Contact( "Blend_T-20".Out_AV_CIP )
   END_RUNG wire#w1
   // the same network as SCL:
   #"AV-20.41"(LOCK := #"lock 1",   // "Valve"
               LIOP_SEL := #init,
               L_AUT := #init,
               L_REMOTE := #init,
               L_RESET := #reset,
               AUT_OP := "Blend_T-20".Out_AV_CIP,
               L_MON := #init,
               INSTANCE := 'AV-20.41',
               QCMD_OP => "AV-20.41");
END_REGION

REGION Network 32: AV-20.42
   RUNG wire#powerrail
      #"AV-20.42"(AUT_OP := wire#w1, LOCK := #"lock 1", ERR_EXTERN :=, LIOP_SEL := #init, L_AUT := #init, L_REMOTE := #init, L_SIM :=, L_RESET := #reset, MAN_OP :=, SIM_OP :=, FB_OPEN :=, FB_CLOSE :=, L_MON := #init, MON_T :=, MON_T_CLOSE :=, INSTANCE := 'AV-20.42', RESTART :=, VISIBILITY :=, OPdwCmd :=, QdwState =>, QwState =>, QCLOSING =>, QCLOSE =>, QOPENING =>, QOPEN =>, QCMD_OP => "AV-20.42", QMON =>, QMON_ERR =>, QMON_T =>, QMON_T_CLOSE =>, QMAN_AUT =>, QREMOTE =>, QSIM =>, QLOCK =>, QERR =>, QERR_EXT =>, QwAlarm =>)
   END_RUNG
   RUNG wire#powerrail
      Contact( "Blend_T-20".Out_AV_CIP )
   END_RUNG wire#w1
   // the same network as SCL:
   #"AV-20.42"(LOCK := #"lock 1",   // "Valve"
               LIOP_SEL := #init,
               L_AUT := #init,
               L_REMOTE := #init,
               L_RESET := #reset,
               AUT_OP := "Blend_T-20".Out_AV_CIP,
               L_MON := #init,
               INSTANCE := 'AV-20.42',
               QCMD_OP => "AV-20.42");
END_REGION
END_FUNCTION_BLOCK

FUNCTION_BLOCK "IO_Valve_Blend21"   // FB25, LAD
{ S7_Optimized_Access := 'FALSE' }
VERSION : 0.1
// stored: AutoNumber true, IsIECCheckEnabled false, SetENOAutomatically false, UDAEnableTagReadback false
   VAR_INPUT
      "lock 1" : Bool;
      "lock 2" : Bool;
      "lock 3" : Bool;
      "lock 4" : Bool;
      init : Bool;
      reset : Bool;
      testing : Bool;
   END_VAR
   VAR
      "AV-21.01" : "Valve";
      "AV-21.02" : "Valve";
      "AV-21.03" : "Valve";
      "AV-21.04" : "Valve";
      "AV-21.05" : "Valve";
      "AV-21.06" : "Valve";
      "AV-21.07" : "Valve";
      "AV-21.08" : "Valve";
      "AV-21.09" : "Valve";
      "AV-21.10" : "Valve";
      "AV-21.11" : "Valve";
      "AV-21.21" : "Valve";
      "AV-21.22" : "Valve";
      "AV-21.23" : "Valve";
      "AV-21.24" : "Valve";
      "AV-21.25" : "Valve";
      "AV-21.26" : "Valve";
      "AV-21.27" : "Valve";
      "AV-21.28" : "Valve";
      "AV-21.29" : "Valve";
      "AV-21.30" : "Valve";
      "AV-21.31" : "Valve";
      "AV-21.32" : "Valve";
      "AV-21.33" : "Valve";
      "AV-21.34" : "Valve";
      "AV-21.35" : "Valve";
      "AV-21.41" : "Valve";
      "AV-21.42" : "Valve";
   END_VAR
BEGIN

REGION Network 1 (SCL): FB OPEN AND CLOSE VALVE T-21
   IF #testing THEN
       // Statement section IF
       #"AV-21.01".FB_OPEN := #"AV-21.01".QCMD_OP;
       #"AV-21.01".FB_CLOSE := NOT #"AV-21.01".QCMD_OP;
       #"AV-21.02".FB_OPEN := #"AV-21.02".QCMD_OP;
       #"AV-21.02".FB_CLOSE := NOT #"AV-21.02".QCMD_OP;
       #"AV-21.03".FB_OPEN := #"AV-21.03".QCMD_OP;
       #"AV-21.03".FB_CLOSE := NOT #"AV-21.03".QCMD_OP;
       #"AV-21.04".FB_OPEN := #"AV-21.04".QCMD_OP;
       #"AV-21.04".FB_CLOSE := NOT #"AV-21.04".QCMD_OP;
       #"AV-21.05".FB_OPEN := #"AV-21.05".QCMD_OP;
       #"AV-21.05".FB_CLOSE := NOT #"AV-21.05".QCMD_OP;
       #"AV-21.06".FB_OPEN := #"AV-21.06".QCMD_OP;
       #"AV-21.06".FB_CLOSE := NOT #"AV-21.06".QCMD_OP;
       #"AV-21.07".FB_OPEN := #"AV-21.07".QCMD_OP;
       #"AV-21.07".FB_CLOSE := NOT #"AV-21.07".QCMD_OP;
       #"AV-21.08".FB_OPEN := #"AV-21.08".QCMD_OP;
       #"AV-21.08".FB_CLOSE := NOT #"AV-21.08".QCMD_OP;
       #"AV-21.09".FB_OPEN := #"AV-21.09".QCMD_OP;
       #"AV-21.09".FB_CLOSE := NOT #"AV-21.09".QCMD_OP;
       #"AV-21.10".FB_OPEN := #"AV-21.10".QCMD_OP;
       #"AV-21.10".FB_CLOSE := NOT #"AV-21.10".QCMD_OP;
       #"AV-21.11".FB_OPEN := #"AV-21.11".QCMD_OP;
       #"AV-21.11".FB_CLOSE := NOT #"AV-21.11".QCMD_OP;
       #"AV-21.21".FB_OPEN := #"AV-21.21".QCMD_OP;
       #"AV-21.21".FB_CLOSE := NOT #"AV-21.21".QCMD_OP;
       #"AV-21.22".FB_OPEN := #"AV-21.22".QCMD_OP;
       #"AV-21.22".FB_CLOSE := NOT #"AV-21.22".QCMD_OP;
       #"AV-21.23".FB_OPEN := #"AV-21.23".QCMD_OP;
       #"AV-21.23".FB_CLOSE := NOT #"AV-21.23".QCMD_OP;
       #"AV-21.24".FB_OPEN := #"AV-21.24".QCMD_OP;
       #"AV-21.24".FB_CLOSE := NOT #"AV-21.24".QCMD_OP;
       #"AV-21.25".FB_OPEN := #"AV-21.25".QCMD_OP;
       #"AV-21.25".FB_CLOSE := NOT #"AV-21.25".QCMD_OP;
       #"AV-21.26".FB_OPEN := #"AV-21.26".QCMD_OP;
       #"AV-21.26".FB_CLOSE := NOT #"AV-21.26".QCMD_OP;
       #"AV-21.27".FB_OPEN := #"AV-21.27".QCMD_OP;
       #"AV-21.27".FB_CLOSE := NOT #"AV-21.27".QCMD_OP;
       #"AV-21.28".FB_OPEN := #"AV-21.28".QCMD_OP;
       #"AV-21.28".FB_CLOSE := NOT #"AV-21.28".QCMD_OP;
       #"AV-21.29".FB_OPEN := #"AV-21.29".QCMD_OP;
       #"AV-21.29".FB_CLOSE := NOT #"AV-21.29".QCMD_OP;
       #"AV-21.30".FB_OPEN := #"AV-21.30".QCMD_OP;
       #"AV-21.30".FB_CLOSE := NOT #"AV-21.30".QCMD_OP;
       #"AV-21.31".FB_OPEN := #"AV-21.31".QCMD_OP;
       #"AV-21.31".FB_CLOSE := NOT #"AV-21.31".QCMD_OP;
       #"AV-21.32".FB_OPEN := #"AV-21.32".QCMD_OP;
       #"AV-21.32".FB_CLOSE := NOT #"AV-21.32".QCMD_OP;
       #"AV-21.33".FB_OPEN := #"AV-21.33".QCMD_OP;
       #"AV-21.33".FB_CLOSE := NOT #"AV-21.33".QCMD_OP;
       #"AV-21.34".FB_OPEN := #"AV-21.34".QCMD_OP;
       #"AV-21.34".FB_CLOSE := NOT #"AV-21.34".QCMD_OP;
       #"AV-21.35".FB_OPEN := #"AV-21.35".QCMD_OP;
       #"AV-21.35".FB_CLOSE := NOT #"AV-21.35".QCMD_OP;
       #"AV-21.41".FB_OPEN := #"AV-21.41".QCMD_OP;
       #"AV-21.41".FB_CLOSE := NOT #"AV-21.41".QCMD_OP;
       #"AV-21.42".FB_OPEN := #"AV-21.42".QCMD_OP;
       #"AV-21.42".FB_CLOSE := NOT #"AV-21.42".QCMD_OP;
   ELSE
       // Statement section ELSE
       #"AV-21.01".FB_OPEN := #"AV-21.01".QCMD_OP;
       #"AV-21.01".FB_CLOSE := NOT #"AV-21.01".QCMD_OP;
       #"AV-21.02".FB_OPEN := NOT "ZSC-21.02";
       #"AV-21.02".FB_CLOSE := "ZSC-21.02";
       #"AV-21.03".FB_OPEN := NOT "ZSC-21.03";
       #"AV-21.03".FB_CLOSE := "ZSC-21.03";
       #"AV-21.04".FB_OPEN := #"AV-21.04".QCMD_OP;
       #"AV-21.04".FB_CLOSE := NOT #"AV-21.04".QCMD_OP;
       #"AV-21.05".FB_OPEN := NOT "ZSC-21.05";
       #"AV-21.05".FB_CLOSE := "ZSC-21.05";
       #"AV-21.06".FB_OPEN := NOT "ZSC-21.06";
       #"AV-21.06".FB_CLOSE := "ZSC-21.06";
       #"AV-21.07".FB_OPEN := #"AV-21.07".QCMD_OP;
       #"AV-21.07".FB_CLOSE := NOT #"AV-21.07".QCMD_OP;
       #"AV-21.08".FB_OPEN := NOT "ZSC-21.08";
       #"AV-21.08".FB_CLOSE := "ZSC-21.08";
       #"AV-21.09".FB_OPEN := NOT "ZSC-21.09";
       #"AV-21.09".FB_CLOSE := "ZSC-21.09";
       #"AV-21.10".FB_OPEN := #"AV-21.10".QCMD_OP;
       #"AV-21.10".FB_CLOSE := NOT #"AV-21.10".QCMD_OP;
       #"AV-21.11".FB_OPEN := NOT "ZSC-21.11";
       #"AV-21.11".FB_CLOSE := "ZSC-21.11";
       #"AV-21.21".FB_OPEN := NOT "ZSC-21.21";
       #"AV-21.21".FB_CLOSE := "ZSC-21.21";
       #"AV-21.22".FB_OPEN := #"AV-21.22".QCMD_OP;
       #"AV-21.22".FB_CLOSE := NOT #"AV-21.22".QCMD_OP;
       #"AV-21.23".FB_OPEN := NOT "ZSC-21.23";
       #"AV-21.23".FB_CLOSE := "ZSC-21.23";
       #"AV-21.24".FB_OPEN := NOT "ZSC-21.24";
       #"AV-21.24".FB_CLOSE := "ZSC-21.24";
       #"AV-21.25".FB_OPEN := NOT "ZSC-21.25";
       #"AV-21.25".FB_CLOSE := "ZSC-21.25";
       #"AV-21.26".FB_OPEN := #"AV-21.26".QCMD_OP;
       #"AV-21.26".FB_CLOSE := NOT #"AV-21.26".QCMD_OP;
       #"AV-21.27".FB_OPEN := NOT "ZSC-21.27";
       #"AV-21.27".FB_CLOSE := "ZSC-21.27";
       #"AV-21.28".FB_OPEN := NOT "ZSC-21.28";
       #"AV-21.28".FB_CLOSE := "ZSC-21.28";
       #"AV-21.29".FB_OPEN := #"AV-21.29".QCMD_OP;
       #"AV-21.29".FB_CLOSE := NOT #"AV-21.29".QCMD_OP;
       #"AV-21.30".FB_OPEN := #"AV-21.30".QCMD_OP;
       #"AV-21.30".FB_CLOSE := NOT #"AV-21.30".QCMD_OP;
       #"AV-21.31".FB_OPEN := NOT "ZSC-21.31";
       #"AV-21.31".FB_CLOSE := "ZSC-21.31";
       #"AV-21.32".FB_OPEN := NOT "ZSC-21.32";
       #"AV-21.32".FB_CLOSE := "ZSC-21.32";
       #"AV-21.33".FB_OPEN := NOT "ZSC-21.33";
       #"AV-21.33".FB_CLOSE := "ZSC-21.33";
       #"AV-21.34".FB_OPEN := NOT "ZSC-21.34";
       #"AV-21.34".FB_CLOSE := "ZSC-21.34";
       #"AV-21.35".FB_OPEN := NOT "ZSC-21.35";
       #"AV-21.35".FB_CLOSE := "ZSC-21.35";
       #"AV-21.41".FB_OPEN := #"AV-21.41".QCMD_OP;
       #"AV-21.41".FB_CLOSE := NOT #"AV-21.41".QCMD_OP;
       #"AV-21.42".FB_OPEN := #"AV-21.42".QCMD_OP;
       #"AV-21.42".FB_CLOSE := NOT #"AV-21.42".QCMD_OP;
   END_IF;
END_REGION

NETWORK
TITLE = FB MONITORING TIME VALVE T-21
// FB OPEN TIME
      L     T#20s;
      T     #"AV-21.01".MON_T;
      T     #"AV-21.02".MON_T;
      T     #"AV-21.03".MON_T;
      T     #"AV-21.04".MON_T;
      T     #"AV-21.05".MON_T;
      T     #"AV-21.06".MON_T;
      T     #"AV-21.07".MON_T;
      T     #"AV-21.08".MON_T;
      T     #"AV-21.09".MON_T;
      T     #"AV-21.10".MON_T;
      T     #"AV-21.11".MON_T;
      T     #"AV-21.21".MON_T;
      T     #"AV-21.22".MON_T;
      T     #"AV-21.23".MON_T;
      T     #"AV-21.24".MON_T;
      T     #"AV-21.25".MON_T;
      T     #"AV-21.26".MON_T;
      T     #"AV-21.27".MON_T;
      T     #"AV-21.28".MON_T;
      T     #"AV-21.29".MON_T;
      T     #"AV-21.30".MON_T;
      T     #"AV-21.31".MON_T;
      T     #"AV-21.32".MON_T;
      T     #"AV-21.33".MON_T;
      T     #"AV-21.34".MON_T;
      T     #"AV-21.35".MON_T;
      T     #"AV-21.41".MON_T;
      T     #"AV-21.42".MON_T;

// FB CLOSE TIME
      L     T#20s;
      T     #"AV-21.01".MON_T_CLOSE;
      T     #"AV-21.02".MON_T_CLOSE;
      T     #"AV-21.03".MON_T_CLOSE;
      T     #"AV-21.04".MON_T_CLOSE;
      T     #"AV-21.05".MON_T_CLOSE;
      T     #"AV-21.06".MON_T_CLOSE;
      T     #"AV-21.07".MON_T_CLOSE;
      T     #"AV-21.08".MON_T_CLOSE;
      T     #"AV-21.09".MON_T_CLOSE;
      T     #"AV-21.10".MON_T_CLOSE;
      T     #"AV-21.11".MON_T_CLOSE;
      T     #"AV-21.21".MON_T_CLOSE;
      T     #"AV-21.22".MON_T_CLOSE;
      T     #"AV-21.23".MON_T_CLOSE;
      T     #"AV-21.24".MON_T_CLOSE;
      T     #"AV-21.25".MON_T_CLOSE;
      T     #"AV-21.26".MON_T_CLOSE;
      T     #"AV-21.27".MON_T_CLOSE;
      T     #"AV-21.28".MON_T_CLOSE;
      T     #"AV-21.29".MON_T_CLOSE;
      T     #"AV-21.30".MON_T_CLOSE;
      T     #"AV-21.31".MON_T_CLOSE;
      T     #"AV-21.32".MON_T_CLOSE;
      T     #"AV-21.33".MON_T_CLOSE;
      T     #"AV-21.34".MON_T_CLOSE;
      T     #"AV-21.35".MON_T_CLOSE;
      T     #"AV-21.41".MON_T_CLOSE;
      T     #"AV-21.42".MON_T_CLOSE;


REGION Network 3: AV-21.01
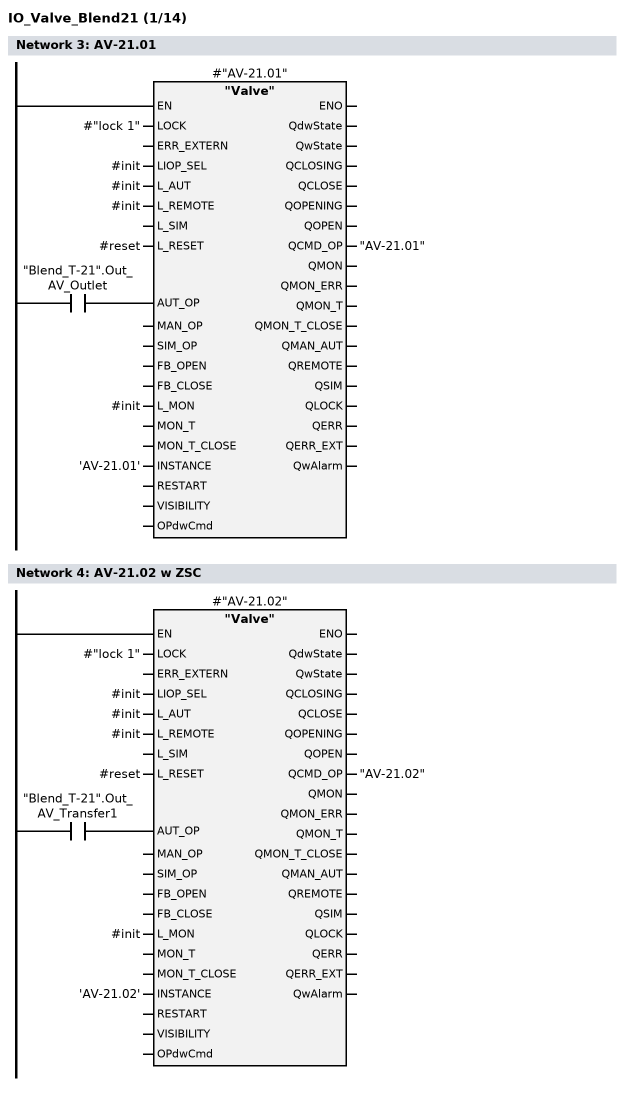
   RUNG wire#powerrail
      #"AV-21.01"(AUT_OP := wire#w1, LOCK := #"lock 1", ERR_EXTERN :=, LIOP_SEL := #init, L_AUT := #init, L_REMOTE := #init, L_SIM :=, L_RESET := #reset, MAN_OP :=, SIM_OP :=, FB_OPEN :=, FB_CLOSE :=, L_MON := #init, MON_T :=, MON_T_CLOSE :=, INSTANCE := 'AV-21.01', RESTART :=, VISIBILITY :=, OPdwCmd :=, QdwState =>, QwState =>, QCLOSING =>, QCLOSE =>, QOPENING =>, QOPEN =>, QCMD_OP => "AV-21.01", QMON =>, QMON_ERR =>, QMON_T =>, QMON_T_CLOSE =>, QMAN_AUT =>, QREMOTE =>, QSIM =>, QLOCK =>, QERR =>, QERR_EXT =>, QwAlarm =>)
   END_RUNG
   RUNG wire#powerrail
      Contact( "Blend_T-21".Out_AV_Outlet )
   END_RUNG wire#w1
   // the same network as SCL:
   #"AV-21.01"(LOCK := #"lock 1",   // "Valve"
               LIOP_SEL := #init,
               L_AUT := #init,
               L_REMOTE := #init,
               L_RESET := #reset,
               AUT_OP := "Blend_T-21".Out_AV_Outlet,
               L_MON := #init,
               INSTANCE := 'AV-21.01',
               QCMD_OP => "AV-21.01");
END_REGION

REGION Network 4: AV-21.02 w ZSC
   RUNG wire#powerrail
      #"AV-21.02"(AUT_OP := wire#w1, LOCK := #"lock 1", ERR_EXTERN :=, LIOP_SEL := #init, L_AUT := #init, L_REMOTE := #init, L_SIM :=, L_RESET := #reset, MAN_OP :=, SIM_OP :=, FB_OPEN :=, FB_CLOSE :=, L_MON := #init, MON_T :=, MON_T_CLOSE :=, INSTANCE := 'AV-21.02', RESTART :=, VISIBILITY :=, OPdwCmd :=, QdwState =>, QwState =>, QCLOSING =>, QCLOSE =>, QOPENING =>, QOPEN =>, QCMD_OP => "AV-21.02", QMON =>, QMON_ERR =>, QMON_T =>, QMON_T_CLOSE =>, QMAN_AUT =>, QREMOTE =>, QSIM =>, QLOCK =>, QERR =>, QERR_EXT =>, QwAlarm =>)
   END_RUNG
   RUNG wire#powerrail
      Contact( "Blend_T-21".Out_AV_Transfer1 )
   END_RUNG wire#w1
   // the same network as SCL:
   #"AV-21.02"(LOCK := #"lock 1",   // "Valve"
               LIOP_SEL := #init,
               L_AUT := #init,
               L_REMOTE := #init,
               L_RESET := #reset,
               AUT_OP := "Blend_T-21".Out_AV_Transfer1,
               L_MON := #init,
               INSTANCE := 'AV-21.02',
               QCMD_OP => "AV-21.02");
END_REGION

REGION Network 5: AV-21.03 w ZSC
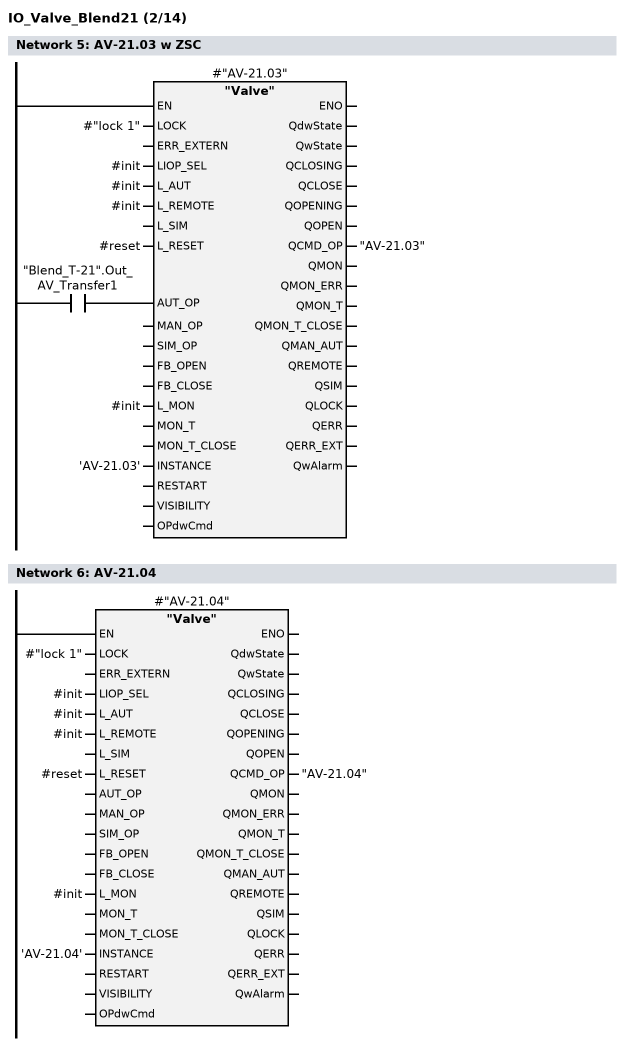
   RUNG wire#powerrail
      #"AV-21.03"(AUT_OP := wire#w1, LOCK := #"lock 1", ERR_EXTERN :=, LIOP_SEL := #init, L_AUT := #init, L_REMOTE := #init, L_SIM :=, L_RESET := #reset, MAN_OP :=, SIM_OP :=, FB_OPEN :=, FB_CLOSE :=, L_MON := #init, MON_T :=, MON_T_CLOSE :=, INSTANCE := 'AV-21.03', RESTART :=, VISIBILITY :=, OPdwCmd :=, QdwState =>, QwState =>, QCLOSING =>, QCLOSE =>, QOPENING =>, QOPEN =>, QCMD_OP => "AV-21.03", QMON =>, QMON_ERR =>, QMON_T =>, QMON_T_CLOSE =>, QMAN_AUT =>, QREMOTE =>, QSIM =>, QLOCK =>, QERR =>, QERR_EXT =>, QwAlarm =>)
   END_RUNG
   RUNG wire#powerrail
      Contact( "Blend_T-21".Out_AV_Transfer1 )
   END_RUNG wire#w1
   // the same network as SCL:
   #"AV-21.03"(LOCK := #"lock 1",   // "Valve"
               LIOP_SEL := #init,
               L_AUT := #init,
               L_REMOTE := #init,
               L_RESET := #reset,
               AUT_OP := "Blend_T-21".Out_AV_Transfer1,
               L_MON := #init,
               INSTANCE := 'AV-21.03',
               QCMD_OP => "AV-21.03");
END_REGION

REGION Network 6: AV-21.04
   RUNG wire#powerrail
      #"AV-21.04"(LOCK := #"lock 1", ERR_EXTERN :=, LIOP_SEL := #init, L_AUT := #init, L_REMOTE := #init, L_SIM :=, L_RESET := #reset, AUT_OP :=, MAN_OP :=, SIM_OP :=, FB_OPEN :=, FB_CLOSE :=, L_MON := #init, MON_T :=, MON_T_CLOSE :=, INSTANCE := 'AV-21.04', RESTART :=, VISIBILITY :=, OPdwCmd :=, QdwState =>, QwState =>, QCLOSING =>, QCLOSE =>, QOPENING =>, QOPEN =>, QCMD_OP => "AV-21.04", QMON =>, QMON_ERR =>, QMON_T =>, QMON_T_CLOSE =>, QMAN_AUT =>, QREMOTE =>, QSIM =>, QLOCK =>, QERR =>, QERR_EXT =>, QwAlarm =>)
   END_RUNG
   // the same network as SCL:
   #"AV-21.04"(LOCK := #"lock 1",   // "Valve"
               LIOP_SEL := #init,
               L_AUT := #init,
               L_REMOTE := #init,
               L_RESET := #reset,
               L_MON := #init,
               INSTANCE := 'AV-21.04',
               QCMD_OP => "AV-21.04");
END_REGION

REGION Network 7: AV-21.05 w ZSC
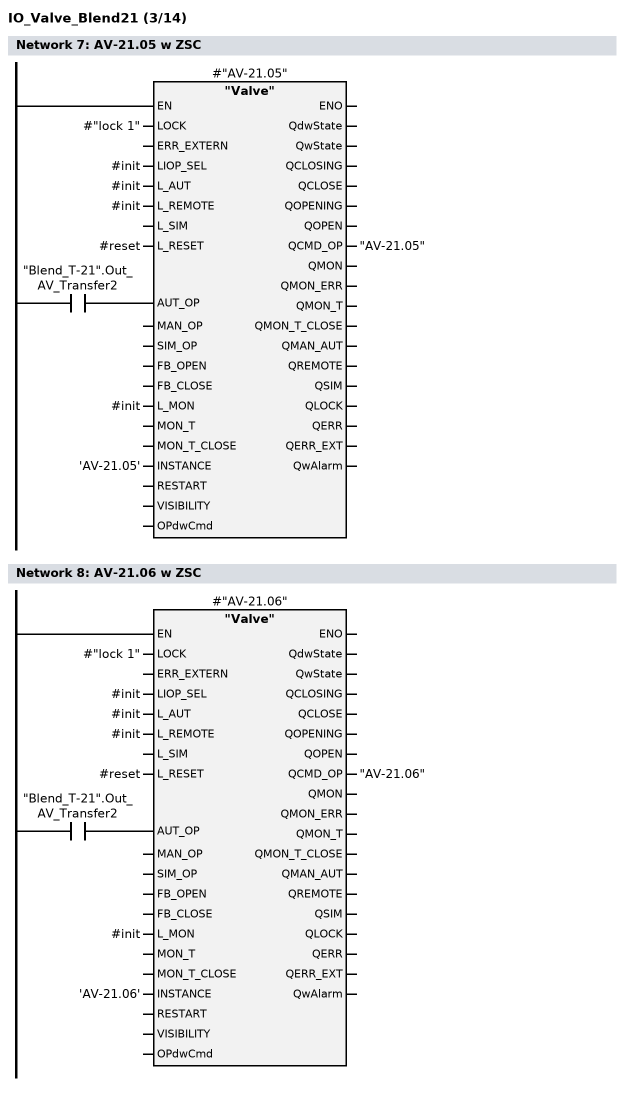
   RUNG wire#powerrail
      #"AV-21.05"(AUT_OP := wire#w1, LOCK := #"lock 1", ERR_EXTERN :=, LIOP_SEL := #init, L_AUT := #init, L_REMOTE := #init, L_SIM :=, L_RESET := #reset, MAN_OP :=, SIM_OP :=, FB_OPEN :=, FB_CLOSE :=, L_MON := #init, MON_T :=, MON_T_CLOSE :=, INSTANCE := 'AV-21.05', RESTART :=, VISIBILITY :=, OPdwCmd :=, QdwState =>, QwState =>, QCLOSING =>, QCLOSE =>, QOPENING =>, QOPEN =>, QCMD_OP => "AV-21.05", QMON =>, QMON_ERR =>, QMON_T =>, QMON_T_CLOSE =>, QMAN_AUT =>, QREMOTE =>, QSIM =>, QLOCK =>, QERR =>, QERR_EXT =>, QwAlarm =>)
   END_RUNG
   RUNG wire#powerrail
      Contact( "Blend_T-21".Out_AV_Transfer2 )
   END_RUNG wire#w1
   // the same network as SCL:
   #"AV-21.05"(LOCK := #"lock 1",   // "Valve"
               LIOP_SEL := #init,
               L_AUT := #init,
               L_REMOTE := #init,
               L_RESET := #reset,
               AUT_OP := "Blend_T-21".Out_AV_Transfer2,
               L_MON := #init,
               INSTANCE := 'AV-21.05',
               QCMD_OP => "AV-21.05");
END_REGION

REGION Network 8: AV-21.06 w ZSC
   RUNG wire#powerrail
      #"AV-21.06"(AUT_OP := wire#w1, LOCK := #"lock 1", ERR_EXTERN :=, LIOP_SEL := #init, L_AUT := #init, L_REMOTE := #init, L_SIM :=, L_RESET := #reset, MAN_OP :=, SIM_OP :=, FB_OPEN :=, FB_CLOSE :=, L_MON := #init, MON_T :=, MON_T_CLOSE :=, INSTANCE := 'AV-21.06', RESTART :=, VISIBILITY :=, OPdwCmd :=, QdwState =>, QwState =>, QCLOSING =>, QCLOSE =>, QOPENING =>, QOPEN =>, QCMD_OP => "AV-21.06", QMON =>, QMON_ERR =>, QMON_T =>, QMON_T_CLOSE =>, QMAN_AUT =>, QREMOTE =>, QSIM =>, QLOCK =>, QERR =>, QERR_EXT =>, QwAlarm =>)
   END_RUNG
   RUNG wire#powerrail
      Contact( "Blend_T-21".Out_AV_Transfer2 )
   END_RUNG wire#w1
   // the same network as SCL:
   #"AV-21.06"(LOCK := #"lock 1",   // "Valve"
               LIOP_SEL := #init,
               L_AUT := #init,
               L_REMOTE := #init,
               L_RESET := #reset,
               AUT_OP := "Blend_T-21".Out_AV_Transfer2,
               L_MON := #init,
               INSTANCE := 'AV-21.06',
               QCMD_OP => "AV-21.06");
END_REGION

REGION Network 9: AV-21.07
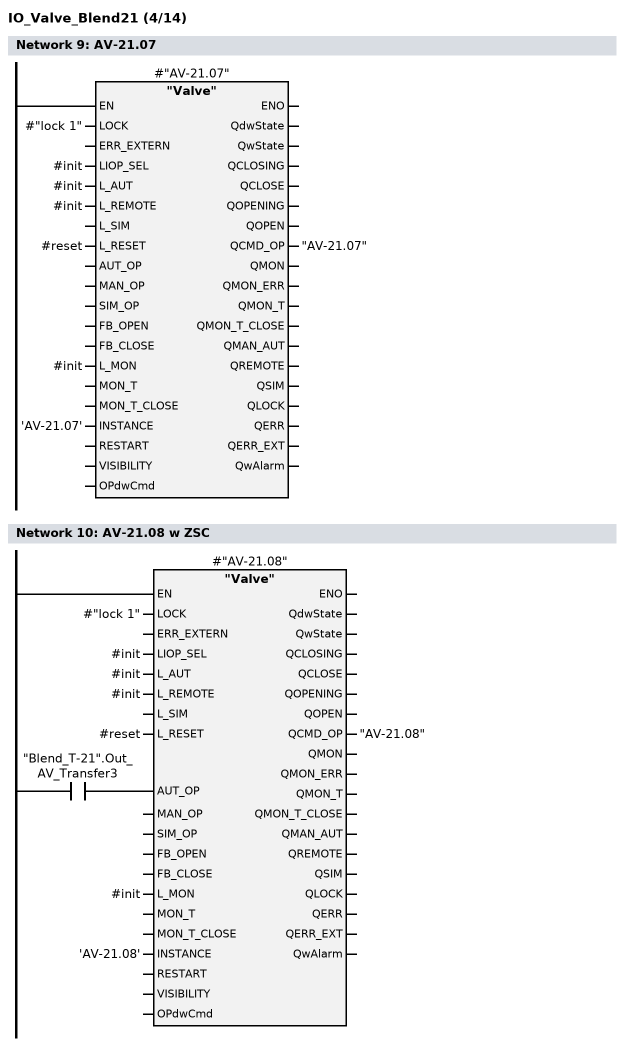
   RUNG wire#powerrail
      #"AV-21.07"(LOCK := #"lock 1", ERR_EXTERN :=, LIOP_SEL := #init, L_AUT := #init, L_REMOTE := #init, L_SIM :=, L_RESET := #reset, AUT_OP :=, MAN_OP :=, SIM_OP :=, FB_OPEN :=, FB_CLOSE :=, L_MON := #init, MON_T :=, MON_T_CLOSE :=, INSTANCE := 'AV-21.07', RESTART :=, VISIBILITY :=, OPdwCmd :=, QdwState =>, QwState =>, QCLOSING =>, QCLOSE =>, QOPENING =>, QOPEN =>, QCMD_OP => "AV-21.07", QMON =>, QMON_ERR =>, QMON_T =>, QMON_T_CLOSE =>, QMAN_AUT =>, QREMOTE =>, QSIM =>, QLOCK =>, QERR =>, QERR_EXT =>, QwAlarm =>)
   END_RUNG
   // the same network as SCL:
   #"AV-21.07"(LOCK := #"lock 1",   // "Valve"
               LIOP_SEL := #init,
               L_AUT := #init,
               L_REMOTE := #init,
               L_RESET := #reset,
               L_MON := #init,
               INSTANCE := 'AV-21.07',
               QCMD_OP => "AV-21.07");
END_REGION

REGION Network 10: AV-21.08 w ZSC
   RUNG wire#powerrail
      #"AV-21.08"(AUT_OP := wire#w1, LOCK := #"lock 1", ERR_EXTERN :=, LIOP_SEL := #init, L_AUT := #init, L_REMOTE := #init, L_SIM :=, L_RESET := #reset, MAN_OP :=, SIM_OP :=, FB_OPEN :=, FB_CLOSE :=, L_MON := #init, MON_T :=, MON_T_CLOSE :=, INSTANCE := 'AV-21.08', RESTART :=, VISIBILITY :=, OPdwCmd :=, QdwState =>, QwState =>, QCLOSING =>, QCLOSE =>, QOPENING =>, QOPEN =>, QCMD_OP => "AV-21.08", QMON =>, QMON_ERR =>, QMON_T =>, QMON_T_CLOSE =>, QMAN_AUT =>, QREMOTE =>, QSIM =>, QLOCK =>, QERR =>, QERR_EXT =>, QwAlarm =>)
   END_RUNG
   RUNG wire#powerrail
      Contact( "Blend_T-21".Out_AV_Transfer3 )
   END_RUNG wire#w1
   // the same network as SCL:
   #"AV-21.08"(LOCK := #"lock 1",   // "Valve"
               LIOP_SEL := #init,
               L_AUT := #init,
               L_REMOTE := #init,
               L_RESET := #reset,
               AUT_OP := "Blend_T-21".Out_AV_Transfer3,
               L_MON := #init,
               INSTANCE := 'AV-21.08',
               QCMD_OP => "AV-21.08");
END_REGION

REGION Network 11: AV-21.09 w ZSC
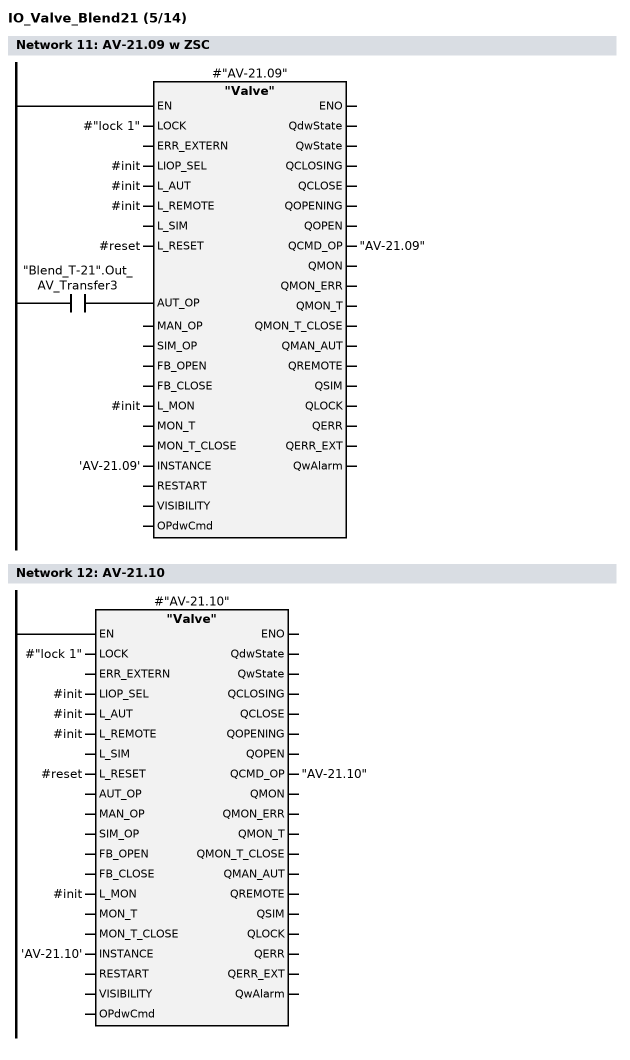
   RUNG wire#powerrail
      #"AV-21.09"(AUT_OP := wire#w1, LOCK := #"lock 1", ERR_EXTERN :=, LIOP_SEL := #init, L_AUT := #init, L_REMOTE := #init, L_SIM :=, L_RESET := #reset, MAN_OP :=, SIM_OP :=, FB_OPEN :=, FB_CLOSE :=, L_MON := #init, MON_T :=, MON_T_CLOSE :=, INSTANCE := 'AV-21.09', RESTART :=, VISIBILITY :=, OPdwCmd :=, QdwState =>, QwState =>, QCLOSING =>, QCLOSE =>, QOPENING =>, QOPEN =>, QCMD_OP => "AV-21.09", QMON =>, QMON_ERR =>, QMON_T =>, QMON_T_CLOSE =>, QMAN_AUT =>, QREMOTE =>, QSIM =>, QLOCK =>, QERR =>, QERR_EXT =>, QwAlarm =>)
   END_RUNG
   RUNG wire#powerrail
      Contact( "Blend_T-21".Out_AV_Transfer3 )
   END_RUNG wire#w1
   // the same network as SCL:
   #"AV-21.09"(LOCK := #"lock 1",   // "Valve"
               LIOP_SEL := #init,
               L_AUT := #init,
               L_REMOTE := #init,
               L_RESET := #reset,
               AUT_OP := "Blend_T-21".Out_AV_Transfer3,
               L_MON := #init,
               INSTANCE := 'AV-21.09',
               QCMD_OP => "AV-21.09");
END_REGION

REGION Network 12: AV-21.10
   RUNG wire#powerrail
      #"AV-21.10"(LOCK := #"lock 1", ERR_EXTERN :=, LIOP_SEL := #init, L_AUT := #init, L_REMOTE := #init, L_SIM :=, L_RESET := #reset, AUT_OP :=, MAN_OP :=, SIM_OP :=, FB_OPEN :=, FB_CLOSE :=, L_MON := #init, MON_T :=, MON_T_CLOSE :=, INSTANCE := 'AV-21.10', RESTART :=, VISIBILITY :=, OPdwCmd :=, QdwState =>, QwState =>, QCLOSING =>, QCLOSE =>, QOPENING =>, QOPEN =>, QCMD_OP => "AV-21.10", QMON =>, QMON_ERR =>, QMON_T =>, QMON_T_CLOSE =>, QMAN_AUT =>, QREMOTE =>, QSIM =>, QLOCK =>, QERR =>, QERR_EXT =>, QwAlarm =>)
   END_RUNG
   // the same network as SCL:
   #"AV-21.10"(LOCK := #"lock 1",   // "Valve"
               LIOP_SEL := #init,
               L_AUT := #init,
               L_REMOTE := #init,
               L_RESET := #reset,
               L_MON := #init,
               INSTANCE := 'AV-21.10',
               QCMD_OP => "AV-21.10");
END_REGION

REGION Network 13: AV-21.11 w ZSC
